C01780=1012.610,-71.664,-108.852,165.899,73.815,164.195
C01781=1012.611,-71.904,-108.833,165.879,73.747,164.164
C01782=1012.612,-72.145,-108.812,165.857,73.678,164.133
C01783=1012.613,-72.385,-108.791,165.837,73.609,164.102
C01784=1012.614,-72.626,-108.771,165.814,73.539,164.070
C01785=1012.614,-72.866,-108.751,165.795,73.470,164.040
C01786=1012.616,-73.107,-108.731,165.775,73.400,164.010
C01787=1012.617,-73.347,-108.710,165.755,73.330,163.979
C01788=1012.617,-73.587,-108.690,165.733,73.259,163.948
C01789=1012.618,-73.827,-108.669,165.715,73.188,163.919
C01790=1012.620,-74.067,-108.649,165.695,73.117,163.888
C01791=1012.621,-74.308,-108.628,165.674,73.045,163.858
C01792=1012.621,-74.547,-108.608,165.656,72.974,163.828
C01793=1012.623,-74.788,-108.588,165.638,72.901,163.799
C01794=1012.623,-75.027,-108.568,165.618,72.829,163.769
C01795=1012.624,-75.267,-108.547,165.599,72.756,163.739
C01796=1012.625,-75.507,-108.526,165.581,72.684,163.710
C01797=1012.627,-75.747,-108.507,165.563,72.611,163.680
C01798=1012.627,-75.987,-108.486,165.543,72.537,163.650
C01799=1012.629,-76.227,-108.465,165.527,72.463,163.622
C01800=1012.630,-76.466,-108.445,165.508,72.389,163.593
C01801=1012.631,-76.706,-108.424,165.491,72.314,163.564
C01802=1012.632,-76.945,-108.404,165.473,72.241,163.535
C01803=1012.633,-77.184,-108.384,165.456,72.165,163.506
C01804=1012.634,-77.424,-108.364,165.438,72.090,163.478
C01805=1012.635,-77.663,-108.344,165.423,72.014,163.450
C01806=1012.637,-77.902,-108.323,165.406,71.939,163.422
C01807=1012.637,-78.141,-108.303,165.390,71.863,163.394
C01808=1012.638,-78.380,-108.283,165.373,71.787,163.365
C01809=1012.640,-78.618,-108.262,165.357,71.711,163.338
C01810=1012.641,-78.857,-108.242,165.342,71.635,163.310
C01811=1012.642,-79.095,-108.222,165.326,71.557,163.282
C01812=1012.643,-79.334,-108.201,165.310,71.481,163.255
C01813=1012.644,-79.572,-108.182,165.296,71.403,163.228
C01814=1012.646,-79.810,-108.161,165.281,71.326,163.201
C01815=1012.647,-80.048,-108.141,165.266,71.248,163.173
C01816=1012.648,-80.341,-108.115,165.248,71.152,163.140
C01817=1012.651,-80.759,-108.080,165.223,71.014,163.093
C01818=1012.652,-80.996,-108.061,165.208,70.935,163.066
C01819=1012.653,-81.232,-108.040,165.194,70.856,163.039
C01820=1012.654,-81.468,-108.020,165.181,70.777,163.013
C01821=1012.656,-81.705,-108.000,165.168,70.698,162.987
C01822=1012.657,-81.943,-107.980,165.153,70.618,162.960
C01823=1012.658,-82.181,-107.959,165.140,70.538,162.934
C01824=1012.660,-82.418,-107.939,165.128,70.458,162.909
C01825=1012.661,-82.653,-107.919,165.116,70.378,162.883
C01826=1012.661,-82.889,-107.899,165.103,70.297,162.857
C01827=1012.664,-83.125,-107.879,165.090,70.217,162.832
C01828=1012.664,-83.361,-107.859,165.078,70.135,162.806
C01829=1012.665,-83.596,-107.840,165.066,70.055,162.781
C01830=1012.667,-83.829,-107.819,165.054,69.974,162.756
C01831=1012.668,-84.062,-107.799,165.043,69.893,162.731
C01832=1012.669,-84.295,-107.780,165.031,69.812,162.706
C01833=1012.671,-84.535,-107.759,165.019,69.728,162.680
C01834=1012.672,-84.792,-107.738,165.008,69.638,162.654
C01835=1012.674,-85.066,-107.714,164.994,69.542,162.625
C01836=1012.676,-85.351,-107.689,164.982,69.441,162.595
C01837=1012.678,-85.634,-107.666,164.969,69.341,162.565
C01838=1012.679,-85.904,-107.643,164.957,69.245,162.538
C01839=1012.681,-86.154,-107.622,164.947,69.156,162.512
C01840=1012.682,-86.389,-107.602,164.937,69.072,162.488
C01841=1012.683,-86.621,-107.582,164.927,68.988,162.464
C01842=1012.685,-86.849,-107.563,164.918,68.905,162.440
C01843=1012.686,-87.073,-107.544,164.910,68.825,162.418
C01844=1012.688,-87.293,-107.525,164.901,68.745,162.396
C01845=1012.689,-87.512,-107.506,164.893,68.665,162.373
C01846=1012.691,-87.727,-107.488,164.884,68.587,162.352
C01847=1012.692,-87.943,-107.470,164.875,68.508,162.329
C01848=1012.693,-88.170,-107.451,164.868,68.424,162.307
C01849=1012.695,-88.397,-107.431,164.860,68.341,162.285
C01850=1012.696,-88.630,-107.411,164.851,68.255,162.261
C01851=1012.698,-88.898,-107.389,164.842,68.156,162.235
C01852=1012.700,-89.194,-107.363,164.832,68.046,162.206
C01853=1012.702,-89.503,-107.337,164.822,67.931,162.175
C01854=1012.704,-89.803,-107.312,164.813,67.819,162.146
C01855=1012.706,-90.082,-107.288,164.804,67.714,162.119
C01856=1012.709,-90.479,-107.254,164.792,67.565,162.080
C01857=1012.711,-90.775,-107.230,164.784,67.452,162.052
C01858=1012.712,-91.025,-107.208,164.778,67.357,162.028
C01859=1012.714,-91.257,-107.188,164.771,67.268,162.006
C01860=1012.716,-91.488,-107.168,164.765,67.180,161.983
C01861=1012.717,-91.720,-107.149,164.760,67.091,161.962
C01862=1012.719,-91.951,-107.129,164.753,67.002,161.940
C01863=1012.721,-92.182,-107.110,164.748,66.913,161.918
C01864=1012.723,-92.412,-107.090,164.742,66.825,161.896
C01865=1012.724,-92.643,-107.070,164.738,66.735,161.875
C01866=1012.726,-92.873,-107.050,164.732,66.645,161.853
C01867=1012.728,-93.103,-107.032,164.726,66.556,161.831
C01868=1012.730,-93.333,-107.012,164.723,66.466,161.811
C01869=1012.731,-93.562,-106.992,164.718,66.377,161.790
C01870=1012.733,-93.790,-106.973,164.714,66.286,161.768
C01871=1012.734,-94.019,-106.953,164.709,66.197,161.747
C01872=1012.737,-94.326,-106.928,164.704,66.075,161.719
C01873=1012.740,-94.702,-106.896,164.697,65.926,161.685
C01874=1012.742,-94.928,-106.877,164.694,65.836,161.664
C01875=1012.743,-95.155,-106.858,164.691,65.746,161.644
C01876=1012.745,-95.381,-106.839,164.687,65.655,161.623
C01877=1012.746,-95.607,-106.819,164.684,65.565,161.604
C01878=1012.748,-95.832,-106.800,164.682,65.475,161.583
C01879=1012.750,-96.057,-106.780,164.679,65.384,161.563
C01880=1012.752,-96.281,-106.762,164.675,65.293,161.543
C01881=1012.754,-96.506,-106.743,164.673,65.203,161.523
C01882=1012.756,-96.730,-106.725,164.671,65.112,161.503
C01883=1012.758,-96.954,-106.705,164.669,65.021,161.484
C01884=1012.760,-97.178,-106.686,164.666,64.929,161.463
C01885=1012.761,-97.401,-106.667,164.664,64.838,161.444
C01886=1012.763,-97.625,-106.648,164.662,64.747,161.424
C01887=1012.766,-97.849,-106.629,164.662,64.655,161.405
C01888=1012.767,-98.072,-106.610,164.660,64.563,161.385
C01889=1012.769,-98.295,-106.591,164.658,64.471,161.366
C01890=1012.771,-98.520,-106.572,164.657,64.378,161.347
C01891=1012.773,-98.744,-106.554,164.655,64.285,161.327
C01892=1012.776,-98.967,-106.534,164.655,64.192,161.308
C01893=1012.777,-99.192,-106.516,164.654,64.099,161.289
C01894=1012.779,-99.416,-106.497,164.653,64.005,161.269
C01895=1012.781,-99.641,-106.477,164.654,63.911,161.251
C01896=1012.783,-99.867,-106.459,164.653,63.817,161.231
C01897=1012.784,-100.092,-106.440,164.653,63.722,161.212
C01898=1012.787,-100.318,-106.421,164.652,63.627,161.193
C01899=1012.789,-100.545,-106.402,164.652,63.532,161.173
C01900=1012.791,-100.771,-106.383,164.652,63.436,161.154
C01901=1012.793,-100.999,-106.364,164.653,63.340,161.135
C01902=1012.796,-101.226,-106.344,164.654,63.244,161.116
C01903=1012.798,-101.454,-106.325,164.655,63.147,161.097
C01904=1012.799,-101.682,-106.305,164.655,63.049,161.078
C01905=1012.802,-101.911,-106.287,164.656,62.952,161.059
C01906=1012.803,-102.140,-106.267,164.658,62.854,161.040
C01907=1012.806,-102.369,-106.248,164.658,62.756,161.021
C01908=1012.808,-102.598,-106.228,164.661,62.658,161.002
C01909=1012.810,-102.827,-106.209,164.661,62.559,160.983
C01910=1012.813,-103.057,-106.189,164.664,62.460,160.964
C01911=1012.814,-103.288,-106.171,164.666,62.361,160.946
C01912=1012.817,-103.517,-106.152,164.667,62.262,160.927
C01913=1012.819,-103.748,-106.132,164.669,62.161,160.908
C01914=1012.821,-103.979,-106.113,164.672,62.062,160.889
C01915=1012.823,-104.209,-106.093,164.674,61.961,160.870
C01916=1012.826,-104.440,-106.074,164.677,61.861,160.852
C01917=1012.829,-104.671,-106.054,164.679,61.760,160.833
C01918=1012.831,-104.902,-106.035,164.682,61.658,160.814
C01919=1012.833,-105.134,-106.016,164.685,61.557,160.796
C01920=1012.836,-105.365,-105.996,164.688,61.456,160.777
C01921=1012.838,-105.597,-105.976,164.693,61.354,160.759
C01922=1012.840,-105.828,-105.957,164.695,61.252,160.740
C01923=1012.842,-106.097,-105.935,164.699,61.134,160.719
C01924=1012.610,-133.983,-104.817,165.422,73.778,163.915
C01925=1012.608,-133.752,-104.837,165.458,73.892,163.966
C01926=1012.607,-133.521,-104.856,165.493,74.006,164.017
C01927=1012.606,-133.290,-104.874,165.530,74.120,164.069
C01928=1012.604,-133.059,-104.894,165.568,74.234,164.122
C01929=1012.602,-132.828,-104.912,165.606,74.346,164.176
C01930=1012.601,-132.597,-104.931,165.646,74.459,164.230
C01931=1012.600,-132.366,-104.949,165.685,74.573,164.284
C01932=1012.597,-132.135,-104.969,165.725,74.685,164.339
C01933=1012.597,-131.904,-104.988,165.766,74.797,164.395
C01934=1012.595,-131.674,-105.007,165.809,74.909,164.452
C01935=1012.594,-131.442,-105.025,165.851,75.020,164.509
C01936=1012.592,-131.211,-105.045,165.895,75.131,164.567
C01937=1012.591,-130.980,-105.063,165.940,75.243,164.626
C01938=1012.589,-130.750,-105.083,165.985,75.355,164.686
C01939=1012.588,-130.519,-105.101,166.032,75.465,164.747
C01940=1012.586,-130.288,-105.120,166.079,75.576,164.808
C01941=1012.585,-130.056,-105.139,166.127,75.687,164.870
C01942=1012.584,-129.825,-105.158,166.176,75.797,164.932
C01943=1012.583,-129.594,-105.177,166.225,75.906,164.996
C01944=1012.581,-129.247,-105.205,166.304,76.071,165.095
C01945=1012.579,-128.901,-105.234,166.382,76.235,165.193
C01946=1012.578,-128.670,-105.253,166.436,76.344,165.260
C01947=1012.576,-128.440,-105.272,166.492,76.453,165.329
C01948=1012.575,-128.208,-105.291,166.546,76.562,165.397
C01949=1012.574,-127.977,-105.310,166.603,76.670,165.467
C01950=1012.573,-127.746,-105.328,166.662,76.778,165.539
C01951=1012.571,-127.515,-105.348,166.722,76.886,165.612
C01952=1012.570,-127.284,-105.367,166.782,76.994,165.684
C01953=1012.569,-127.053,-105.386,166.845,77.102,165.760
C01954=1012.568,-126.822,-105.405,166.906,77.209,165.834
C01955=1012.567,-126.590,-105.424,166.970,77.317,165.911
C01956=1012.565,-126.360,-105.443,167.038,77.424,165.990
C01957=1012.564,-126.129,-105.462,167.104,77.531,166.069
C01958=1012.563,-125.898,-105.481,167.171,77.638,166.149
C01959=1012.562,-125.667,-105.501,167.239,77.743,166.229
C01960=1012.561,-125.435,-105.520,167.312,77.850,166.313
C01961=1012.559,-125.204,-105.538,167.384,77.955,166.397
C01962=1012.559,-124.973,-105.557,167.456,78.062,166.482
C01963=1012.558,-124.742,-105.576,167.532,78.168,166.570
C01964=1012.557,-124.511,-105.595,167.607,78.273,166.657
C01965=1012.556,-124.280,-105.614,167.687,78.379,166.748
C01966=1012.555,-124.050,-105.633,167.768,78.483,166.840
C01967=1012.554,-123.818,-105.652,167.849,78.588,166.933
C01968=1012.553,-123.587,-105.671,167.930,78.693,167.026
C01969=1012.552,-123.355,-105.690,168.017,78.798,167.124
C01970=1012.551,-123.125,-105.709,168.102,78.902,167.221
C01971=1012.550,-122.893,-105.728,168.191,79.006,167.321
C01972=1012.549,-122.662,-105.747,168.280,79.109,167.421
C01973=1012.548,-122.431,-105.767,168.372,79.214,167.524
C01974=1012.547,-122.200,-105.786,168.465,79.317,167.629
C01975=1012.546,-121.968,-105.804,168.561,79.420,167.735
C01976=1012.545,-121.737,-105.825,168.659,79.524,167.845
C01977=1012.543,-121.507,-105.843,168.760,79.627,167.956
C01978=1012.542,-121.275,-105.862,168.862,79.729,168.068
C01979=1012.542,-121.045,-105.882,168.968,79.832,168.185
C01980=1012.541,-120.813,-105.900,169.074,79.935,168.302
C01981=1012.540,-120.583,-105.920,169.185,80.037,168.422
C01982=1012.539,-120.351,-105.939,169.294,80.139,168.542
C01983=1012.539,-120.119,-105.958,169.410,80.241,168.668
C01984=1012.538,-119.888,-105.978,169.524,80.343,168.794
C01985=1012.537,-119.657,-105.996,169.644,80.444,168.923
C01986=1012.536,-119.426,-106.015,169.766,80.545,169.055
C01987=1012.535,-119.195,-106.035,169.889,80.646,169.188
C01988=1012.534,-118.963,-106.054,170.018,80.747,169.327
C01989=1012.533,-118.732,-106.073,170.147,80.847,169.466
C01990=1012.533,-118.501,-106.092,170.280,80.948,169.609
C01991=1012.531,-118.092,-106.126,170.523,81.125,169.870
C01992=1012.530,-117.807,-106.150,170.698,81.249,170.056
C01993=1012.529,-117.576,-106.169,170.847,81.348,170.215
C01994=1012.530,-117.345,-106.188,170.996,81.448,170.373
C01995=1012.529,-117.114,-106.206,171.150,81.547,170.537
C01996=1012.528,-116.883,-106.226,171.308,81.647,170.704
C01997=1012.527,-116.651,-106.245,171.467,81.745,170.872
C01998=1012.526,-116.420,-106.264,171.635,81.844,171.049
C01999=1012.526,-116.189,-106.284,171.803,81.942,171.227
C02000=1012.525,-115.958,-106.303,171.976,82.041,171.408
C02001=1012.524,-115.727,-106.322,172.154,82.139,171.596
C02002=1012.524,-115.495,-106.341,172.334,82.237,171.785
C02003=1012.523,-115.264,-106.361,172.524,82.334,171.983
C02004=1012.522,-115.033,-106.380,172.715,82.431,172.183
C02005=1012.522,-114.801,-106.399,172.911,82.529,172.388
C02006=1012.521,-114.570,-106.419,173.118,82.626,172.603
C02007=1012.520,-114.338,-106.437,173.323,82.722,172.817
C02008=1012.520,-114.107,-106.457,173.538,82.819,173.040
C02009=1012.519,-113.876,-106.476,173.759,82.916,173.270
C02010=1012.518,-113.645,-106.496,173.984,83.012,173.503
C02011=1012.518,-113.413,-106.515,174.216,83.107,173.743
C02012=1012.517,-113.181,-106.534,174.453,83.203,173.990
C02013=1012.517,-112.950,-106.554,174.700,83.298,174.245
C02014=1012.516,-112.719,-106.573,174.955,83.394,174.507
C02015=1012.515,-112.488,-106.592,175.212,83.488,174.773
C02016=1012.515,-112.256,-106.611,175.484,83.583,175.052
C02017=1012.515,-112.025,-106.630,175.758,83.677,175.335
C02018=1012.514,-111.793,-106.650,176.042,83.771,175.627
C02019=1012.514,-111.563,-106.669,176.336,83.865,175.928
C02020=1012.513,-111.330,-106.688,176.634,83.957,176.234
C02021=1012.512,-111.099,-106.707,176.948,84.051,176.556
C02022=1012.512,-110.868,-106.727,177.266,84.144,176.882
C02023=1012.511,-110.636,-106.746,177.597,84.236,177.220
C02024=1012.511,-110.405,-106.766,177.939,84.327,177.569
C02025=1012.511,-110.173,-106.785,178.292,84.420,177.931
C02026=1012.510,-109.942,-106.805,178.660,84.511,178.305
C02027=1012.510,-109.710,-106.824,179.033,84.602,178.686
C02028=1012.509,-109.479,-106.843,179.420,84.692,179.080
C02029=1012.509,-109.245,-106.863,179.828,84.783,179.496
C02030=1012.508,-109.004,-106.883,-179.733,84.876,179.941
C02031=1012.508,-108.754,-106.904,-179.271,84.972,-179.589
C02032=1012.508,-108.493,-106.926,-178.768,85.072,-179.077
C02033=1012.507,-108.225,-106.948,-178.225,85.174,-178.527
C02034=1012.507,-107.951,-106.971,-177.642,85.279,-177.936
C02035=1012.506,-107.674,-106.994,-177.040,85.382,-177.326
C02036=1012.505,-107.399,-107.017,-176.409,85.485,-176.686
C02037=1012.505,-107.129,-107.041,-175.756,85.585,-176.026
C02038=1012.505,-106.867,-107.062,-175.101,85.681,-175.363
C02039=1012.504,-106.614,-107.083,-174.437,85.773,-174.692
C02040=1012.504,-106.372,-107.104,-173.774,85.861,-174.022
C02041=1012.504,-106.136,-107.124,-173.103,85.946,-173.345
C02042=1012.503,-105.758,-107.155,-171.968,86.080,-172.200
C02043=1012.503,-105.442,-107.182,-170.971,86.189,-171.195
C02044=1012.503,-105.210,-107.201,-170.188,86.270,-170.405
C02045=1012.502,-104.979,-107.220,-169.382,86.349,-169.594
C02046=1012.502,-104.748,-107.240,-168.553,86.427,-168.758
C02047=1012.501,-104.516,-107.259,-167.673,86.504,-167.872
C02048=1012.501,-104.286,-107.278,-166.751,86.580,-166.944
C02049=1012.501,-104.054,-107.298,-165.803,86.655,-165.991
C02050=1012.502,-103.825,-107.318,-164.808,86.729,-164.990
C02051=1012.501,-103.594,-107.337,-163.769,86.801,-163.945
C02052=1012.500,-103.364,-107.356,-162.680,86.872,-162.851
C02053=1012.501,-103.134,-107.376,-161.552,86.943,-161.717
C02054=1012.499,-102.904,-107.395,-160.379,87.011,-160.538
C02055=1012.500,-102.675,-107.415,-159.145,87.078,-159.299
C02056=1012.500,-102.445,-107.434,-157.853,87.143,-158.001
C02057=1012.499,-102.216,-107.453,-156.504,87.207,-156.647
C02058=1012.499,-101.987,-107.473,-155.105,87.269,-155.242
C02059=1012.499,-101.759,-107.491,-153.627,87.329,-153.759
C02060=1012.499,-101.531,-107.511,-152.100,87.387,-152.227
C02061=1012.499,-101.303,-107.530,-150.532,87.442,-150.654
C02062=1012.499,-101.076,-107.550,-148.865,87.496,-148.982
C02063=1012.498,-100.849,-107.568,-147.155,87.547,-147.268
C02064=1012.499,-100.621,-107.587,-145.373,87.596,-145.481
C02065=1012.498,-100.396,-107.607,-143.518,87.642,-143.620
C02066=1012.498,-100.170,-107.626,-141.589,87.686,-141.687
C02067=1012.498,-99.944,-107.645,-139.610,87.726,-139.703
C02068=1012.498,-99.719,-107.664,-137.573,87.764,-137.661
C02069=1012.498,-99.494,-107.683,-135.467,87.798,-135.551
C02070=1012.498,-99.270,-107.701,-133.296,87.830,-133.376
C02071=1012.497,-99.045,-107.721,-131.089,87.858,-131.163
C02072=1012.497,-98.822,-107.740,-128.799,87.883,-128.869
C02073=1012.497,-98.597,-107.759,-126.499,87.904,-126.565
C02074=1012.497,-98.373,-107.778,-124.139,87.922,-124.200
C02075=1012.497,-98.150,-107.796,-121.757,87.935,-121.814
C02076=1012.497,-97.926,-107.815,-119.371,87.946,-119.424
C02077=1012.498,-97.703,-107.834,-116.939,87.953,-116.988
C02078=1012.497,-97.479,-107.853,-114.519,87.956,-114.563
C02079=1012.497,-97.256,-107.872,-112.071,87.955,-112.112
C02080=1012.497,-97.032,-107.891,-109.652,87.951,-109.688
C02081=1012.497,-96.808,-107.909,-107.246,87.943,-107.278
C02082=1012.497,-96.584,-107.929,-104.882,87.931,-104.911
C02083=1012.497,-96.360,-107.947,-102.528,87.916,-102.553
C02084=1012.496,-96.135,-107.967,-100.232,87.897,-100.252
C02085=1012.496,-95.910,-107.986,-97.978,87.875,-97.995
C02086=1012.497,-95.686,-108.005,-95.754,87.850,-95.767
C02087=1012.497,-95.460,-108.024,-93.602,87.822,-93.611
C02088=1012.497,-95.234,-108.044,-91.510,87.790,-91.516
C02089=1012.497,-95.007,-108.062,-89.460,87.756,-89.462
C02090=1012.497,-94.781,-108.081,-87.490,87.719,-87.488
C02091=1012.496,-94.553,-108.101,-85.584,87.679,-85.578
C02092=1012.497,-94.326,-108.120,-83.748,87.637,-83.739
C02093=1012.497,-94.098,-108.139,-81.974,87.592,-81.961
C02094=1012.497,-93.869,-108.158,-80.253,87.545,-80.237
C02095=1012.497,-93.641,-108.178,-78.611,87.496,-78.591
C02096=1012.496,-93.412,-108.198,-77.048,87.446,-77.026
C02097=1012.497,-93.182,-108.217,-75.532,87.393,-75.505
C02098=1012.497,-92.952,-108.237,-74.077,87.338,-74.047
C02099=1012.498,-92.598,-108.267,-71.951,87.251,-71.916
C02100=1012.497,-92.261,-108.295,-70.074,87.165,-70.034
C02101=1012.498,-92.030,-108.315,-68.844,87.104,-68.801
C02102=1012.497,-91.799,-108.334,-67.684,87.043,-67.639
C02103=1012.498,-91.568,-108.354,-66.554,86.980,-66.505
C02104=1012.497,-91.337,-108.374,-65.488,86.917,-65.436
C02105=1012.497,-91.105,-108.393,-64.449,86.851,-64.394
C02106=1012.498,-90.855,-108.414,-63.392,86.780,-63.334
C02107=1012.498,-90.558,-108.440,-62.190,86.694,-62.129
C02108=1012.498,-90.162,-108.474,-60.695,86.579,-60.628
C02109=1012.498,-89.884,-108.497,-59.706,86.496,-59.637
C02110=1012.498,-89.582,-108.523,-58.692,86.406,-58.619
C02111=1012.498,-89.274,-108.549,-57.706,86.313,-57.630
C02112=1012.499,-88.978,-108.574,-56.802,86.222,-56.722
C02113=1012.499,-88.710,-108.597,-56.028,86.140,-55.945
C02114=1012.500,-88.477,-108.617,-55.388,86.068,-55.302
C02115=1012.500,-88.251,-108.636,-54.781,85.998,-54.693
C02116=1012.499,-88.025,-108.655,-54.206,85.928,-54.116
C02117=1012.500,-87.808,-108.674,-53.669,85.860,-53.576
C02118=1012.500,-87.592,-108.692,-53.150,85.792,-53.055
C02119=1012.500,-87.373,-108.711,-52.646,85.723,-52.550
C02120=1012.501,-87.154,-108.730,-52.159,85.653,-52.061
C02121=1012.500,-86.931,-108.748,-51.673,85.582,-51.572
C02122=1012.500,-86.701,-108.768,-51.201,85.510,-51.098
C02123=1012.501,-86.470,-108.787,-50.737,85.436,-50.633
C02124=1012.501,-86.236,-108.808,-50.281,85.361,-50.174
C02125=1012.502,-85.985,-108.829,-49.812,85.281,-49.702
C02126=1012.502,-85.715,-108.852,-49.331,85.196,-49.219
C02127=1012.502,-85.433,-108.876,-48.840,85.105,-48.727
C02128=1012.502,-85.148,-108.900,-48.368,85.014,-48.252
C02129=1012.503,-84.872,-108.924,-47.926,84.925,-47.807
C02130=1012.503,-84.617,-108.945,-47.534,84.842,-47.414
C02131=1012.503,-84.376,-108.966,-47.173,84.765,-47.051
C02132=1012.503,-84.143,-108.986,-46.839,84.690,-46.715
C02133=1012.504,-83.911,-109.006,-46.514,84.616,-46.388
C02134=1012.504,-83.678,-109.026,-46.199,84.540,-46.072
C02135=1012.504,-83.443,-109.046,-45.892,84.465,-45.763
C02136=1012.504,-83.207,-109.066,-45.589,84.389,-45.459
C02137=1012.504,-82.970,-109.086,-45.299,84.313,-45.167
C02138=1012.505,-82.735,-109.106,-45.012,84.237,-44.878
C02139=1012.505,-82.499,-109.126,-44.737,84.161,-44.602
C02140=1012.505,-82.262,-109.146,-44.470,84.086,-44.333
C02141=1012.505,-82.025,-109.167,-44.209,84.010,-44.071
C02142=1012.506,-81.787,-109.186,-43.956,83.933,-43.816
C02143=1012.506,-81.551,-109.207,-43.709,83.857,-43.568
C02144=1012.507,-81.314,-109.226,-43.468,83.781,-43.326
C02145=1012.507,-81.078,-109.248,-43.237,83.705,-43.094
C02146=1012.508,-80.841,-109.267,-43.011,83.630,-42.867
C02147=1012.508,-80.604,-109.288,-42.787,83.554,-42.641
C02148=1012.508,-80.368,-109.308,-42.572,83.479,-42.426
C02149=1012.508,-80.130,-109.328,-42.363,83.403,-42.215
C02150=1012.508,-79.893,-109.348,-42.158,83.327,-42.010
C02151=1012.509,-79.654,-109.369,-41.958,83.253,-41.808
C02152=1012.509,-79.416,-109.389,-41.762,83.177,-41.612
C02153=1012.510,-79.178,-109.410,-41.575,83.102,-41.423
C02154=1012.510,-78.940,-109.430,-41.388,83.026,-41.236
C02155=1012.511,-78.701,-109.450,-41.209,82.951,-41.056
C02156=1012.511,-78.463,-109.470,-41.030,82.876,-40.876
C02157=1012.511,-78.223,-109.491,-40.858,82.801,-40.703
C02158=1012.511,-77.985,-109.511,-40.690,82.726,-40.535
C02159=1012.512,-77.746,-109.531,-40.525,82.651,-40.369
C02160=1012.512,-77.443,-109.557,-40.322,82.557,-40.165
C02161=1012.513,-77.029,-109.592,-40.054,82.428,-39.896
C02162=1012.513,-76.789,-109.613,-39.906,82.354,-39.747
C02163=1012.514,-76.550,-109.633,-39.760,82.280,-39.601
C02164=1012.514,-76.310,-109.654,-39.618,82.206,-39.458
C02165=1012.515,-76.071,-109.674,-39.478,82.132,-39.318
C02166=1012.515,-75.831,-109.695,-39.340,82.058,-39.179
C02167=1012.515,-75.590,-109.716,-39.205,81.984,-39.044
C02168=1012.516,-75.352,-109.736,-39.075,81.911,-38.914
C02169=1012.516,-75.111,-109.757,-38.945,81.838,-38.783
C02170=1012.516,-74.871,-109.777,-38.820,81.765,-38.658
C02171=1012.517,-74.631,-109.797,-38.698,81.692,-38.535
C02172=1012.517,-74.392,-109.818,-38.576,81.620,-38.413
C02173=1012.517,-74.151,-109.839,-38.458,81.546,-38.295
C02174=1012.518,-73.912,-109.859,-38.344,81.475,-38.181
C02175=1012.518,-73.671,-109.879,-38.229,81.402,-38.065
C02176=1012.519,-73.431,-109.900,-38.119,81.331,-37.955
C02177=1012.520,-73.191,-109.920,-38.011,81.259,-37.847
C02178=1012.519,-72.951,-109.941,-37.905,81.187,-37.741
C02179=1012.520,-72.710,-109.961,-37.801,81.115,-37.637
C02180=1012.520,-72.470,-109.982,-37.700,81.045,-37.536
C02181=1012.521,-72.230,-110.002,-37.598,80.973,-37.433
C02182=1012.522,-71.989,-110.023,-37.501,80.902,-37.337
C02183=1012.522,-71.748,-110.043,-37.405,80.831,-37.242
C02184=1012.522,-71.508,-110.064,-37.310,80.762,-37.145
C02185=1012.523,-71.267,-110.085,-37.217,80.691,-37.053
C02186=1012.523,-71.027,-110.106,-37.125,80.620,-36.962
C02187=1012.524,-70.787,-110.126,-37.037,80.551,-36.873
C02188=1012.525,-70.546,-110.146,-36.950,80.482,-36.786
C02189=1012.525,-70.305,-110.166,-36.861,80.412,-36.698
C02190=1012.525,-70.064,-110.187,-36.779,80.343,-36.617
C02191=1012.525,-69.824,-110.208,-36.696,80.274,-36.534
C02192=1012.526,-69.583,-110.229,-36.614,80.205,-36.452
C02193=1012.526,-69.343,-110.249,-36.535,80.137,-36.373
C02194=1012.527,-69.101,-110.270,-36.454,80.068,-36.292
C02195=1012.527,-68.861,-110.290,-36.378,79.999,-36.217
C02196=1012.528,-68.620,-110.310,-36.302,79.931,-36.142
C02197=1012.528,-68.380,-110.331,-36.229,79.865,-36.068
C02198=1012.529,-68.139,-110.352,-36.155,79.797,-35.995
C02199=1012.529,-67.899,-110.373,-36.085,79.729,-35.926
C02200=1012.529,-67.658,-110.393,-36.014,79.663,-35.855
C02201=1012.530,-67.417,-110.413,-35.944,79.596,-35.786
C02202=1012.531,-67.177,-110.433,-35.876,79.530,-35.718
C02203=1012.531,-66.936,-110.454,-35.808,79.463,-35.651
C02204=1012.531,-66.696,-110.475,-35.744,79.397,-35.587
C02205=1012.532,-66.455,-110.496,-35.677,79.331,-35.520
C02206=1012.533,-66.215,-110.516,-35.614,79.265,-35.458
C02207=1012.533,-65.976,-110.537,-35.553,79.201,-35.398
C02208=1012.533,-65.735,-110.557,-35.491,79.135,-35.336
C02209=1012.534,-65.495,-110.578,-35.429,79.070,-35.275
C02210=1012.534,-65.255,-110.598,-35.370,79.006,-35.217
C02211=1012.535,-65.016,-110.619,-35.311,78.942,-35.159
C02212=1012.535,-64.776,-110.639,-35.254,78.877,-35.103
C02213=1012.536,-64.536,-110.659,-35.199,78.814,-35.048
C02214=1012.536,-64.297,-110.680,-35.142,78.750,-34.992
C02215=1012.537,-64.058,-110.700,-35.088,78.687,-34.939
C02216=1012.537,-63.819,-110.720,-35.033,78.625,-34.884
C02217=1012.537,-63.580,-110.741,-34.980,78.562,-34.833
C02218=1012.538,-63.341,-110.762,-34.927,78.499,-34.780
C02219=1012.539,-63.102,-110.782,-34.877,78.437,-34.732
C02220=1012.539,-62.864,-110.802,-34.827,78.375,-34.682
C02221=1012.540,-62.625,-110.823,-34.777,78.313,-34.634
C02222=1012.540,-62.387,-110.843,-34.727,78.253,-34.584
C02223=1012.540,-62.149,-110.863,-34.679,78.191,-34.537
C02224=1012.541,-61.910,-110.884,-34.632,78.131,-34.490
C02225=1012.541,-61.673,-110.904,-34.585,78.070,-34.445
C02226=1012.542,-61.436,-110.924,-34.539,78.010,-34.399
C02227=1012.542,-61.198,-110.944,-34.494,77.950,-34.355
C02228=1012.543,-60.961,-110.964,-34.450,77.890,-34.313
C02229=1012.543,-60.724,-110.985,-34.405,77.831,-34.268
C02230=1012.544,-60.487,-111.005,-34.361,77.772,-34.225
C02231=1012.544,-60.250,-111.025,-34.318,77.713,-34.183
C02232=1012.545,-60.014,-111.045,-34.277,77.655,-34.143
C02233=1012.546,-59.778,-111.065,-34.235,77.597,-34.102
C02234=1012.546,-59.541,-111.085,-34.195,77.539,-34.064
C02235=1012.546,-59.305,-111.105,-34.155,77.481,-34.024
C02236=1012.547,-58.914,-111.139,-34.089,77.386,-33.960
C02237=1012.548,-58.599,-111.166,-34.037,77.310,-33.909
C02238=1012.548,-58.364,-111.186,-34.000,77.254,-33.873
C02239=1012.549,-58.129,-111.206,-33.963,77.197,-33.838
C02240=1012.549,-57.894,-111.226,-33.927,77.142,-33.803
C02241=1012.550,-57.659,-111.246,-33.890,77.086,-33.767
C02242=1012.550,-57.425,-111.266,-33.854,77.031,-33.732
C02243=1012.551,-57.190,-111.286,-33.819,76.976,-33.699
C02244=1012.551,-56.956,-111.306,-33.785,76.921,-33.665
C02245=1012.552,-56.722,-111.326,-33.750,76.866,-33.632
C02246=1012.552,-56.488,-111.346,-33.717,76.813,-33.600
C02247=1012.553,-56.254,-111.366,-33.682,76.758,-33.566
C02248=1012.553,-56.020,-111.385,-33.651,76.704,-33.536
C02249=1012.553,-55.786,-111.405,-33.618,76.650,-33.505
C02250=1012.554,-55.553,-111.425,-33.586,76.598,-33.474
C02251=1012.555,-55.319,-111.445,-33.554,76.545,-33.443
C02252=1012.554,-55.085,-111.465,-33.524,76.492,-33.415
C02253=1012.555,-54.851,-111.485,-33.493,76.440,-33.385
C02254=1012.556,-54.618,-111.505,-33.463,76.388,-33.355
///RCONF 0,0,0,0,1,0,0,0,0,0,0,0,0,0,0,0,0,0,0,0,0,0,0,0
C02255=1012.557,-54.384,-111.525,-33.432,76.336,-33.326
C02256=1012.556,-54.151,-111.545,-33.402,76.284,-33.297
C02257=1012.557,-53.917,-111.564,-33.374,76.233,-33.270
C02258=1012.558,-53.684,-111.584,-33.344,76.180,-33.242
C02259=1012.558,-53.450,-111.604,-33.315,76.130,-33.214
C02260=1012.559,-53.216,-111.625,-33.289,76.079,-33.189
C02261=1012.559,-52.982,-111.644,-33.260,76.029,-33.162
C02262=1012.560,-52.749,-111.664,-33.232,75.978,-33.135
C02263=1012.561,-52.515,-111.684,-33.206,75.928,-33.110
C02264=1012.560,-52.282,-111.704,-33.179,75.879,-33.085
C02265=1012.561,-52.048,-111.723,-33.153,75.829,-33.060
C02266=1012.561,-51.814,-111.743,-33.126,75.780,-33.034
C02267=1012.562,-51.581,-111.763,-33.100,75.731,-33.008
C02268=1012.562,-51.347,-111.784,-33.075,75.682,-32.986
C02269=1012.563,-51.113,-111.803,-33.051,75.634,-32.963
C02270=1012.564,-50.879,-111.823,-33.025,75.585,-32.937
C02271=1012.564,-50.646,-111.844,-33.000,75.536,-32.914
C02272=1012.564,-50.412,-111.863,-32.976,75.490,-32.891
C02273=1012.564,-50.179,-111.882,-32.952,75.441,-32.869
C02274=1012.565,-49.945,-111.902,-32.928,75.395,-32.846
C02275=1012.565,-49.711,-111.923,-32.906,75.347,-32.826
C02276=1012.566,-49.477,-111.942,-32.883,75.300,-32.804
C02277=1012.567,-49.244,-111.962,-32.859,75.253,-32.782
C02278=1012.567,-49.010,-111.983,-32.837,75.207,-32.760
C02279=1012.567,-48.776,-112.002,-32.814,75.162,-32.739
C02280=1012.568,-48.542,-112.022,-32.792,75.115,-32.717
C02281=1012.569,-48.309,-112.042,-32.770,75.070,-32.696
C02282=1012.569,-48.074,-112.062,-32.749,75.024,-32.677
C02283=1012.569,-47.842,-112.081,-32.728,74.979,-32.658
C02284=1012.570,-47.608,-112.101,-32.706,74.934,-32.638
C02285=1012.569,-47.374,-112.121,-32.686,74.890,-32.619
C02286=1012.570,-47.140,-112.141,-32.665,74.846,-32.599
C02287=1012.571,-46.907,-112.161,-32.645,74.801,-32.581
C02288=1012.571,-46.672,-112.181,-32.625,74.757,-32.562
C02289=1012.571,-46.439,-112.201,-32.605,74.713,-32.543
C02290=1012.572,-46.205,-112.221,-32.586,74.670,-32.525
C02291=1012.572,-45.971,-112.240,-32.565,74.627,-32.505
C02292=1012.573,-45.737,-112.260,-32.546,74.584,-32.488
C02293=1012.573,-45.503,-112.280,-32.527,74.541,-32.470
C02294=1012.573,-45.269,-112.300,-32.509,74.500,-32.453
C02295=1012.574,-45.036,-112.320,-32.490,74.457,-32.436
C02296=1012.575,-44.802,-112.339,-32.472,74.415,-32.419
C02297=1012.575,-44.568,-112.360,-32.454,74.374,-32.402
C02298=1012.575,-44.334,-112.379,-32.437,74.332,-32.387
C02299=1012.575,-44.100,-112.400,-32.418,74.291,-32.369
C02300=1012.576,-43.866,-112.419,-32.401,74.250,-32.352
C02301=1012.577,-43.632,-112.439,-32.384,74.209,-32.338
C02302=1012.576,-43.398,-112.459,-32.366,74.169,-32.320
C02303=1012.577,-43.164,-112.479,-32.349,74.128,-32.305
C02304=1012.578,-42.931,-112.499,-32.332,74.089,-32.289
C02305=1012.578,-42.696,-112.519,-32.317,74.050,-32.275
C02306=1012.579,-42.463,-112.538,-32.300,74.010,-32.259
C02307=1012.578,-42.228,-112.558,-32.284,73.971,-32.245
C02308=1012.579,-41.995,-112.578,-32.269,73.932,-32.231
C02309=1012.579,-41.760,-112.598,-32.252,73.894,-32.215
C02310=1012.579,-41.526,-112.617,-32.237,73.854,-32.202
C02311=1012.580,-41.293,-112.637,-32.221,73.816,-32.186
C02312=1012.581,-41.057,-112.657,-32.206,73.779,-32.173
C02313=1012.581,-40.824,-112.677,-32.191,73.741,-32.159
C02314=1012.581,-40.589,-112.697,-32.176,73.704,-32.146
C02315=1012.582,-40.356,-112.717,-32.162,73.666,-32.132
C02316=1012.582,-40.122,-112.737,-32.146,73.630,-32.117
C02317=1012.583,-39.888,-112.757,-32.132,73.592,-32.104
C02318=1012.583,-39.654,-112.776,-32.117,73.557,-32.091
C02319=1012.583,-39.419,-112.796,-32.104,73.520,-32.080
C02320=1012.584,-39.186,-112.816,-32.090,73.484,-32.067
C02321=1012.584,-38.951,-112.836,-32.076,73.448,-32.054
C02322=1012.585,-38.717,-112.856,-32.062,73.414,-32.041
C02323=1012.585,-38.483,-112.876,-32.049,73.378,-32.028
C02324=1012.585,-38.249,-112.895,-32.036,73.343,-32.017
C02325=1012.585,-38.015,-112.916,-32.022,73.308,-32.005
C02326=1012.586,-37.781,-112.935,-32.009,73.274,-31.992
C02327=1012.586,-37.547,-112.956,-31.996,73.240,-31.979
C02328=1012.586,-37.313,-112.975,-31.983,73.206,-31.969
C02329=1012.587,-37.078,-112.995,-31.970,73.172,-31.956
C02330=1012.587,-36.844,-113.015,-31.958,73.139,-31.946
C02331=1012.587,-36.610,-113.035,-31.946,73.105,-31.935
C02332=1012.588,-36.375,-113.054,-31.934,73.073,-31.924
C02333=1012.588,-36.142,-113.075,-31.921,73.040,-31.912
C02334=1012.588,-35.908,-113.094,-31.910,73.008,-31.903
C02335=1012.588,-35.673,-113.114,-31.898,72.975,-31.891
C02336=1012.589,-35.439,-113.134,-31.886,72.943,-31.880
C02337=1012.589,-35.204,-113.154,-31.874,72.912,-31.868
C02338=1012.590,-34.970,-113.173,-31.864,72.881,-31.860
C02339=1012.590,-34.736,-113.194,-31.851,72.850,-31.848
C02340=1012.590,-34.502,-113.213,-31.841,72.818,-31.839
C02341=1012.590,-34.268,-113.233,-31.830,72.788,-31.829
C02342=1012.591,-34.034,-113.253,-31.819,72.758,-31.818
C02343=1012.591,-33.799,-113.273,-31.808,72.727,-31.808
C02344=1012.591,-33.565,-113.293,-31.797,72.697,-31.798
C02345=1012.592,-33.331,-113.313,-31.787,72.667,-31.790
C02346=1012.591,-33.097,-113.332,-31.776,72.639,-31.779
C02347=1012.592,-32.863,-113.352,-31.766,72.609,-31.771
C02348=1012.592,-32.628,-113.371,-31.756,72.580,-31.761
C02349=1012.592,-32.395,-113.391,-31.745,72.551,-31.751
C02350=1012.592,-32.160,-113.411,-31.736,72.523,-31.744
C02351=1012.593,-31.925,-113.431,-31.725,72.495,-31.732
C02352=1012.593,-31.692,-113.451,-31.716,72.467,-31.724
C02353=1012.594,-31.457,-113.471,-31.706,72.439,-31.716
C02354=1012.594,-31.223,-113.490,-31.696,72.412,-31.706
C02355=1012.594,-30.989,-113.510,-31.688,72.384,-31.699
C02356=1012.594,-30.755,-113.530,-31.678,72.357,-31.689
C02357=1012.594,-30.521,-113.550,-31.668,72.331,-31.681
C02358=1012.595,-30.286,-113.569,-31.659,72.304,-31.672
C02359=1012.595,-30.053,-113.590,-31.650,72.278,-31.664
C02360=1012.595,-29.818,-113.609,-31.642,72.252,-31.658
C02361=1012.595,-29.583,-113.629,-31.633,72.226,-31.649
C02362=1012.596,-29.350,-113.649,-31.624,72.201,-31.641
C02363=1012.596,-29.134,-113.667,-31.616,72.178,-31.633
C02364=1012.597,-28.881,-113.688,-31.608,72.151,-31.626
C02365=1012.596,-28.647,-113.708,-31.599,72.126,-31.618
C02366=1012.596,-28.413,-113.729,-31.590,72.101,-31.610
C02367=1012.597,-28.179,-113.748,-31.583,72.077,-31.603
C02368=1012.597,-27.944,-113.768,-31.574,72.054,-31.595
C02369=1012.597,-27.711,-113.788,-31.567,72.030,-31.588
C02370=1012.597,-27.476,-113.808,-31.558,72.007,-31.580
C02371=1012.598,-27.242,-113.827,-31.551,71.983,-31.573
C02372=1012.597,-27.008,-113.847,-31.543,71.960,-31.567
C02373=1012.598,-26.774,-113.867,-31.535,71.937,-31.558
C02374=1012.598,-26.540,-113.886,-31.528,71.915,-31.552
C02375=1012.598,-26.305,-113.906,-31.520,71.892,-31.545
C02376=1012.599,-26.072,-113.926,-31.512,71.871,-31.537
C02377=1012.598,-25.837,-113.946,-31.506,71.849,-31.532
C02378=1012.599,-25.603,-113.965,-31.498,71.827,-31.524
C02379=1012.599,-25.369,-113.986,-31.492,71.806,-31.519
C02380=1012.599,-25.135,-114.005,-31.485,71.785,-31.512
C02381=1012.599,-24.901,-114.025,-31.478,71.764,-31.505
C02382=1012.599,-24.666,-114.045,-31.471,71.743,-31.498
C02383=1012.600,-24.433,-114.065,-31.464,71.724,-31.492
C02384=1012.599,-24.198,-114.085,-31.457,71.703,-31.485
C02385=1012.600,-23.964,-114.104,-31.451,71.683,-31.480
C02386=1012.600,-23.730,-114.124,-31.444,71.664,-31.473
C02387=1012.601,-23.496,-114.144,-31.438,71.646,-31.468
C02388=1012.600,-23.262,-114.163,-31.432,71.626,-31.463
C02389=1012.601,-23.028,-114.183,-31.425,71.607,-31.454
C02390=1012.600,-22.795,-114.203,-31.419,71.589,-31.449
C02391=1012.600,-22.560,-114.223,-31.413,71.570,-31.444
C02392=1012.601,-22.326,-114.242,-31.407,71.552,-31.439
C02393=1012.601,-22.092,-114.262,-31.401,71.534,-31.432
C02394=1012.601,-21.858,-114.282,-31.396,71.517,-31.428
C02395=1012.601,-21.624,-114.301,-31.389,71.499,-31.421
C02396=1012.602,-21.390,-114.321,-31.384,71.482,-31.416
C02397=1012.601,-21.156,-114.341,-31.378,71.466,-31.410
C02398=1012.601,-20.921,-114.361,-31.372,71.449,-31.405
C02399=1012.602,-20.688,-114.381,-31.368,71.433,-31.401
C02400=1012.601,-20.454,-114.401,-31.361,71.417,-31.394
C02401=1012.602,-20.176,-114.423,-31.355,71.398,-31.388
C02402=1012.602,-19.826,-114.453,-31.347,71.374,-31.380
C02403=1012.601,-19.565,-114.475,-31.342,71.358,-31.375
C02404=1012.602,-19.266,-114.501,-31.335,71.338,-31.368
C02405=1012.602,-18.940,-114.528,-31.329,71.317,-31.362
C02406=1012.602,-18.609,-114.557,-31.322,71.298,-31.356
C02407=1012.602,-18.291,-114.583,-31.316,71.279,-31.349
C02408=1012.602,-18.007,-114.607,-31.310,71.262,-31.344
C02409=1012.602,-17.759,-114.628,-31.305,71.249,-31.339
C02410=1012.602,-17.528,-114.648,-31.300,71.235,-31.333
C02411=1012.602,-17.297,-114.667,-31.297,71.223,-31.330
C02412=1012.602,-17.063,-114.686,-31.292,71.210,-31.326
C02413=1012.602,-16.826,-114.707,-31.288,71.197,-31.322
C02414=1012.602,-16.589,-114.726,-31.284,71.185,-31.317
C02415=1012.603,-16.354,-114.746,-31.279,71.173,-31.312
C02416=1012.603,-16.119,-114.766,-31.276,71.161,-31.309
C02417=1012.602,-15.883,-114.786,-31.271,71.150,-31.304
C02418=1012.602,-15.647,-114.806,-31.267,71.138,-31.300
C02419=1012.603,-15.414,-114.825,-31.263,71.127,-31.296
C02420=1012.602,-15.185,-114.845,-31.260,71.117,-31.293
C02421=1012.603,-14.957,-114.864,-31.256,71.106,-31.288
C02422=1012.603,-14.733,-114.883,-31.252,71.096,-31.284
C02423=1012.602,-14.510,-114.902,-31.249,71.087,-31.280
C02424=1012.602,-14.287,-114.921,-31.245,71.078,-31.276
C02425=1012.603,-14.063,-114.939,-31.242,71.069,-31.273
C02426=1012.603,-13.837,-114.959,-31.238,71.059,-31.268
C02427=1012.602,-13.608,-114.978,-31.235,71.051,-31.265
C02428=1012.603,-13.375,-114.998,-31.232,71.042,-31.262
C02429=1012.602,-13.138,-115.017,-31.229,71.033,-31.258
C02430=1012.602,-12.897,-115.038,-31.226,71.024,-31.255
C02431=1012.602,-12.652,-115.058,-31.223,71.015,-31.252
C02432=1012.602,-12.407,-115.079,-31.219,71.008,-31.247
C02433=1012.602,-12.160,-115.100,-31.216,70.999,-31.244
C02434=1012.603,-11.913,-115.120,-31.213,70.992,-31.241
C02435=1012.602,-11.666,-115.141,-31.210,70.983,-31.238
C02436=1012.601,-11.418,-115.162,-31.208,70.976,-31.234
C02437=1012.602,-11.169,-115.183,-31.205,70.968,-31.231
C02438=1012.602,-10.920,-115.204,-31.202,70.961,-31.227
C02439=1012.602,-10.671,-115.226,-31.198,70.955,-31.222
C02440=1012.601,-10.421,-115.247,-31.196,70.949,-31.220
C02441=1012.602,-10.171,-115.267,-31.193,70.943,-31.217
C02442=1012.601,-9.921,-115.289,-31.191,70.937,-31.215
C02443=1012.601,-9.669,-115.309,-31.189,70.931,-31.211
C02444=1012.601,-9.418,-115.331,-31.186,70.926,-31.207
C02445=1012.601,-9.167,-115.352,-31.183,70.920,-31.204
C02446=1012.601,-8.916,-115.373,-31.181,70.915,-31.201
C02447=1012.600,-8.665,-115.394,-31.179,70.911,-31.199
C02448=1012.601,-8.413,-115.416,-31.177,70.907,-31.195
C02449=1012.601,-8.161,-115.437,-31.175,70.902,-31.193
C02450=1012.600,-7.909,-115.458,-31.173,70.899,-31.191
C02451=1012.601,-7.655,-115.480,-31.171,70.895,-31.187
C02452=1012.600,-7.401,-115.500,-31.169,70.892,-31.184
C02453=1012.600,-7.146,-115.523,-31.167,70.889,-31.182
C02454=1012.600,-6.889,-115.544,-31.165,70.886,-31.179
C02455=1012.599,-6.633,-115.565,-31.163,70.883,-31.175
C02456=1012.600,-6.375,-115.587,-31.162,70.881,-31.174
C02457=1012.599,-6.117,-115.609,-31.160,70.879,-31.171
C02458=1012.599,-5.859,-115.630,-31.159,70.878,-31.168
C02459=1012.599,-5.601,-115.652,-31.158,70.876,-31.167
C02460=1012.599,-5.344,-115.674,-31.156,70.875,-31.163
C02461=1012.599,-5.092,-115.695,-31.155,70.874,-31.162
C02462=1012.598,-4.848,-115.716,-31.154,70.874,-31.160
C02463=1012.598,-4.613,-115.736,-31.153,70.873,-31.159
C02464=1012.598,-4.384,-115.754,-31.152,70.873,-31.156
C02465=1012.598,-4.158,-115.773,-31.150,70.873,-31.153
C02466=1012.598,-3.932,-115.793,-31.149,70.872,-31.151
C02467=1012.597,-3.702,-115.812,-31.149,70.873,-31.150
C02468=1012.597,-3.465,-115.833,-31.148,70.874,-31.148
C02469=1012.598,-3.222,-115.852,-31.147,70.875,-31.147
C02470=1012.597,-2.978,-115.873,-31.146,70.877,-31.143
C02471=1012.597,-2.733,-115.894,-31.146,70.878,-31.143
C02472=1012.597,-2.489,-115.914,-31.145,70.879,-31.141
C02473=1012.596,-2.246,-115.934,-31.145,70.882,-31.139
C02474=1012.597,-2.003,-115.955,-31.144,70.884,-31.138
C02475=1012.596,-1.761,-115.975,-31.144,70.887,-31.136
C02476=1012.595,-1.519,-115.996,-31.143,70.889,-31.134
C02477=1012.595,-1.279,-116.016,-31.143,70.892,-31.132
C02478=1012.595,-1.039,-116.037,-31.143,70.895,-31.131
C02479=1012.595,-0.800,-116.056,-31.143,70.899,-31.131
C02480=1012.594,-0.561,-116.076,-31.143,70.903,-31.129
C02481=1012.594,-0.323,-116.096,-31.143,70.906,-31.128
C02482=1012.594,-0.087,-116.116,-31.143,70.910,-31.126
C02483=1012.594,0.149,-116.136,-31.142,70.914,-31.124
C02484=1012.593,0.384,-116.156,-31.143,70.918,-31.125
C02485=1012.593,0.618,-116.175,-31.143,70.923,-31.123
C02486=1012.593,0.852,-116.195,-31.143,70.928,-31.122
C02487=1012.592,1.089,-116.215,-31.143,70.933,-31.119
C02488=1012.592,1.326,-116.235,-31.143,70.938,-31.119
C02489=1012.592,1.562,-116.255,-31.145,70.944,-31.119
C02490=1012.592,1.796,-116.274,-31.144,70.950,-31.117
C02491=1012.591,2.025,-116.294,-31.146,70.955,-31.118
C02492=1012.591,2.246,-116.313,-31.145,70.961,-31.115
C02493=1012.590,2.655,-116.346,-31.147,70.972,-31.115
C02494=1012.590,3.039,-116.379,-31.148,70.983,-31.113
C02495=1012.589,3.431,-116.412,-31.150,70.996,-31.113
C02496=1012.589,3.639,-116.430,-31.150,71.002,-31.112
C02497=1012.589,3.857,-116.448,-31.152,71.009,-31.112
C02498=1012.588,4.086,-116.467,-31.152,71.018,-31.111
C02499=1012.588,4.319,-116.486,-31.154,71.025,-31.111
C02500=1012.588,4.552,-116.507,-31.154,71.033,-31.110
C02501=1012.587,4.784,-116.526,-31.156,71.042,-31.110
C02502=1012.587,5.014,-116.545,-31.156,71.050,-31.109
C02503=1012.587,5.246,-116.564,-31.158,71.059,-31.109
C02504=1012.586,5.479,-116.584,-31.159,71.068,-31.109
C02505=1012.586,5.711,-116.603,-31.160,71.078,-31.108
C02506=1012.586,5.946,-116.623,-31.162,71.087,-31.108
C02507=1012.585,6.180,-116.643,-31.163,71.098,-31.108
C02508=1012.585,6.413,-116.663,-31.166,71.107,-31.109
C02509=1012.584,6.646,-116.682,-31.167,71.117,-31.108
C02510=1012.584,6.877,-116.701,-31.168,71.128,-31.107
C02511=1012.583,7.106,-116.721,-31.171,71.137,-31.109
C02512=1012.584,7.333,-116.740,-31.172,71.148,-31.109
C02513=1012.583,7.560,-116.758,-31.174,71.158,-31.109
C02514=1012.583,7.786,-116.777,-31.176,71.170,-31.110
C02515=1012.582,8.009,-116.796,-31.177,71.181,-31.108
C02516=1012.582,8.233,-116.815,-31.179,71.192,-31.108
C02517=1012.582,8.455,-116.834,-31.181,71.203,-31.110
C02518=1012.581,8.678,-116.853,-31.184,71.215,-31.111
C02519=1012.581,8.900,-116.871,-31.186,71.227,-31.111
C02520=1012.581,9.123,-116.890,-31.188,71.239,-31.110
C02521=1012.580,9.346,-116.909,-31.190,71.250,-31.112
C02522=1012.580,9.568,-116.927,-31.192,71.263,-31.111
C02523=1012.580,9.792,-116.946,-31.194,71.275,-31.112
C02524=1012.579,10.015,-116.965,-31.196,71.288,-31.112
C02525=1012.578,10.239,-116.984,-31.199,71.301,-31.113
C02526=1012.579,10.465,-117.003,-31.202,71.314,-31.114
C02527=1012.577,10.689,-117.022,-31.204,71.327,-31.115
C02528=1012.577,10.910,-117.041,-31.206,71.340,-31.115
C02529=1012.576,11.128,-117.058,-31.209,71.353,-31.116
C02530=1012.576,11.344,-117.076,-31.212,71.367,-31.119
C02531=1012.577,11.560,-117.095,-31.214,71.381,-31.118
C02532=1012.575,11.779,-117.113,-31.217,71.394,-31.119
C02533=1012.575,12.003,-117.132,-31.220,71.409,-31.120
C02534=1012.575,12.229,-117.151,-31.224,71.424,-31.122
C02535=1012.574,12.459,-117.170,-31.226,71.438,-31.123
C02536=1012.574,12.687,-117.189,-31.229,71.455,-31.124
C02537=1012.574,12.915,-117.209,-31.232,71.469,-31.125
C02538=1012.573,13.144,-117.228,-31.235,71.486,-31.126
C02539=1012.572,13.372,-117.248,-31.239,71.501,-31.128
C02540=1012.572,13.599,-117.266,-31.242,71.517,-31.129
C02541=1012.571,13.827,-117.285,-31.246,71.534,-31.131
C02542=1012.571,14.053,-117.304,-31.250,71.549,-31.133
C02543=1012.571,14.279,-117.323,-31.253,71.566,-31.134
C02544=1012.570,14.506,-117.342,-31.257,71.583,-31.136
C02545=1012.570,14.733,-117.361,-31.260,71.601,-31.137
C02546=1012.569,14.958,-117.380,-31.264,71.617,-31.139
C02547=1012.568,15.185,-117.399,-31.268,71.634,-31.141
C02548=1012.567,15.411,-117.418,-31.271,71.652,-31.142
C02549=1012.567,15.637,-117.437,-31.275,71.669,-31.144
C02550=1012.567,15.864,-117.456,-31.279,71.688,-31.146
C02551=1012.566,16.091,-117.474,-31.282,71.706,-31.147
C02552=1012.566,16.319,-117.494,-31.287,71.723,-31.150
C02553=1012.565,16.546,-117.514,-31.291,71.742,-31.153
C02554=1012.564,16.775,-117.533,-31.295,71.762,-31.154
C02555=1012.564,17.004,-117.552,-31.299,71.781,-31.156
C02556=1012.564,17.234,-117.571,-31.304,71.800,-31.159
C02557=1012.563,17.464,-117.590,-31.308,71.820,-31.160
C02558=1012.562,17.695,-117.610,-31.313,71.839,-31.164
C02559=1012.562,17.927,-117.629,-31.317,71.859,-31.166
C02560=1012.561,18.159,-117.648,-31.322,71.880,-31.169
C02561=1012.561,18.392,-117.668,-31.327,71.901,-31.171
C02562=1012.560,18.626,-117.688,-31.332,71.921,-31.175
C02563=1012.560,18.859,-117.707,-31.337,71.942,-31.178
C02564=1012.559,19.121,-117.730,-31.343,71.967,-31.181
C02565=1012.558,19.426,-117.755,-31.349,71.994,-31.184
C02566=1012.557,19.822,-117.787,-31.358,72.032,-31.190
C02567=1012.557,20.122,-117.813,-31.365,72.060,-31.194
C02568=1012.556,20.441,-117.840,-31.372,72.090,-31.198
C02569=1012.555,20.760,-117.866,-31.379,72.122,-31.202
C02570=1012.554,21.070,-117.893,-31.388,72.152,-31.207
C02571=1012.553,21.359,-117.917,-31.394,72.181,-31.212
C02572=1012.553,21.618,-117.939,-31.400,72.207,-31.215
C02573=1012.552,22.029,-117.973,-31.411,72.248,-31.222
C02574=1012.551,22.442,-118.008,-31.422,72.291,-31.228
C02575=1012.549,22.787,-118.036,-31.431,72.327,-31.235
C02576=1012.549,23.078,-118.061,-31.439,72.358,-31.241
C02577=1012.549,23.379,-118.086,-31.448,72.390,-31.246
C02578=1012.547,23.743,-118.116,-31.458,72.430,-31.253
C02579=1012.546,24.109,-118.147,-31.468,72.469,-31.259
C02580=1012.545,24.406,-118.172,-31.477,72.503,-31.265
C02581=1012.544,24.642,-118.192,-31.483,72.529,-31.268
C02582=1012.543,24.878,-118.212,-31.490,72.556,-31.273
C02583=1012.543,25.114,-118.231,-31.497,72.582,-31.278
C02584=1012.542,25.349,-118.251,-31.505,72.609,-31.283
C02585=1012.541,25.585,-118.271,-31.513,72.636,-31.290
C02586=1012.541,25.823,-118.291,-31.519,72.663,-31.293
C02587=1012.541,26.060,-118.311,-31.527,72.692,-31.298
C02588=1012.540,26.296,-118.331,-31.535,72.719,-31.305
C02589=1012.539,26.533,-118.350,-31.542,72.747,-31.310
C02590=1012.538,26.768,-118.369,-31.550,72.775,-31.315
C02591=1012.537,27.003,-118.390,-31.558,72.803,-31.320
C02592=1012.537,27.237,-118.409,-31.565,72.832,-31.325
C02593=1012.536,27.471,-118.429,-31.574,72.861,-31.332
C02594=1012.536,27.705,-118.448,-31.581,72.889,-31.337
C02595=1012.535,27.938,-118.468,-31.590,72.918,-31.344
C02596=1012.534,28.173,-118.488,-31.598,72.947,-31.349
C02597=1012.534,28.407,-118.507,-31.607,72.976,-31.356
C02598=1012.533,28.642,-118.526,-31.615,73.006,-31.361
C02599=1012.532,28.876,-118.547,-31.624,73.035,-31.368
C02600=1012.532,29.112,-118.566,-31.633,73.066,-31.375
C02601=1012.530,29.347,-118.586,-31.642,73.096,-31.381
C02602=1012.530,29.583,-118.605,-31.650,73.126,-31.387
C02603=1012.529,29.818,-118.625,-31.659,73.156,-31.394
C02604=1012.528,30.053,-118.645,-31.668,73.187,-31.401
C02605=1012.528,30.288,-118.664,-31.678,73.219,-31.408
C02606=1012.527,30.524,-118.684,-31.687,73.250,-31.415
C02607=1012.526,30.759,-118.703,-31.696,73.282,-31.422
C02608=1012.525,30.994,-118.724,-31.706,73.312,-31.429
C02609=1012.525,31.229,-118.743,-31.715,73.344,-31.436
C02610=1012.524,31.465,-118.763,-31.725,73.376,-31.443
C02611=1012.524,31.700,-118.782,-31.735,73.409,-31.451
C02612=1012.522,31.936,-118.802,-31.745,73.441,-31.459
C02613=1012.521,32.170,-118.822,-31.755,73.474,-31.467
C02614=1012.521,32.406,-118.842,-31.766,73.506,-31.476
C02615=1012.520,32.642,-118.862,-31.777,73.539,-31.485
C02616=1012.519,32.877,-118.881,-31.786,73.572,-31.491
C02617=1012.518,33.112,-118.900,-31.797,73.605,-31.500
C02618=1012.518,33.346,-118.920,-31.808,73.639,-31.509
C02619=1012.517,33.583,-118.940,-31.818,73.673,-31.516
C02620=1012.516,33.818,-118.960,-31.830,73.706,-31.526
C02621=1012.515,34.053,-118.979,-31.841,73.740,-31.535
C02622=1012.514,34.288,-118.999,-31.852,73.775,-31.545
C02623=1012.514,34.524,-119.018,-31.863,73.810,-31.552
C02624=1012.513,34.759,-119.039,-31.875,73.845,-31.562
C02625=1012.513,34.994,-119.058,-31.886,73.879,-31.571
C02626=1012.511,35.229,-119.078,-31.897,73.914,-31.579
C02627=1012.511,35.466,-119.098,-31.910,73.950,-31.591
C02628=1012.510,35.701,-119.117,-31.921,73.985,-31.599
C02629=1012.509,35.936,-119.136,-31.934,74.020,-31.610
C02630=1012.508,36.171,-119.156,-31.946,74.056,-31.620
C02631=1012.508,36.407,-119.176,-31.959,74.092,-31.630
C02632=1012.507,36.642,-119.196,-31.971,74.128,-31.640
C02633=1012.506,36.877,-119.215,-31.984,74.165,-31.652
C02634=1012.505,37.112,-119.235,-31.997,74.201,-31.662
C02635=1012.504,37.349,-119.255,-32.010,74.238,-31.672
C02636=1012.504,37.584,-119.274,-32.022,74.274,-31.682
C02637=1012.502,37.819,-119.294,-32.035,74.312,-31.693
C02638=1012.502,38.054,-119.313,-32.049,74.349,-31.705
C02639=1012.501,38.290,-119.333,-32.063,74.387,-31.717
C02640=1012.500,38.525,-119.353,-32.076,74.425,-31.728
C02641=1012.500,38.760,-119.373,-32.090,74.462,-31.738
C02642=1012.498,38.995,-119.392,-32.104,74.501,-31.751
C02643=1012.498,39.232,-119.412,-32.118,74.539,-31.763
C02644=1012.497,39.467,-119.431,-32.133,74.577,-31.776
C02645=1012.496,39.702,-119.451,-32.148,74.616,-31.789
C02646=1012.495,39.937,-119.470,-32.162,74.655,-31.800
C02647=1012.495,40.173,-119.490,-32.176,74.693,-31.813
C02648=1012.493,40.409,-119.510,-32.192,74.733,-31.826
C02649=1012.493,40.644,-119.529,-32.206,74.772,-31.838
C02650=1012.491,40.879,-119.549,-32.222,74.811,-31.853
C02651=1012.491,41.115,-119.569,-32.238,74.851,-31.866
C02652=1012.490,41.350,-119.588,-32.253,74.891,-31.879
C02653=1012.489,41.586,-119.608,-32.269,74.931,-31.893
C02654=1012.488,41.821,-119.628,-32.286,74.971,-31.908
C02655=1012.488,42.057,-119.647,-32.301,75.012,-31.920
C02656=1012.487,42.292,-119.667,-32.318,75.053,-31.936
C02657=1012.485,42.527,-119.687,-32.334,75.094,-31.950
C02658=1012.485,42.763,-119.707,-32.350,75.134,-31.964
C02659=1012.484,42.998,-119.726,-32.367,75.176,-31.979
C02660=1012.483,43.234,-119.746,-32.385,75.218,-31.995
C02661=1012.482,43.469,-119.765,-32.403,75.258,-32.011
C02662=1012.482,43.705,-119.785,-32.420,75.300,-32.026
C02663=1012.480,43.940,-119.805,-32.438,75.342,-32.042
C02664=1012.479,44.176,-119.825,-32.455,75.385,-32.057
C02665=1012.479,44.411,-119.844,-32.474,75.427,-32.074
C02666=1012.478,44.647,-119.864,-32.493,75.469,-32.091
C02667=1012.477,44.882,-119.884,-32.510,75.512,-32.107
C02668=1012.476,45.117,-119.903,-32.529,75.554,-32.124
C02669=1012.475,45.353,-119.923,-32.549,75.598,-32.141
C02670=1012.474,45.589,-119.942,-32.567,75.641,-32.157
C02671=1012.473,45.824,-119.961,-32.587,75.684,-32.177
C02672=1012.472,46.061,-119.981,-32.607,75.728,-32.195
C02673=1012.471,46.296,-120.001,-32.627,75.771,-32.213
C02674=1012.470,46.531,-120.020,-32.647,75.815,-32.231
C02675=1012.470,46.767,-120.040,-32.666,75.860,-32.248
C02676=1012.469,47.003,-120.060,-32.687,75.903,-32.267
C02677=1012.467,47.238,-120.079,-32.709,75.948,-32.287
C02678=1012.467,47.474,-120.099,-32.730,75.993,-32.306
C02679=1012.466,47.709,-120.118,-32.749,76.037,-32.324
C02680=1012.465,47.945,-120.138,-32.772,76.082,-32.345
C02681=1012.464,48.181,-120.158,-32.793,76.127,-32.364
C02682=1012.464,48.416,-120.177,-32.816,76.173,-32.386
C02683=1012.462,48.651,-120.197,-32.838,76.218,-32.406
C02684=1012.461,48.887,-120.217,-32.861,76.264,-32.428
C02685=1012.460,49.123,-120.236,-32.884,76.309,-32.448
C02686=1012.460,49.358,-120.255,-32.907,76.355,-32.471
C02687=1012.459,49.594,-120.275,-32.930,76.402,-32.491
C02688=1012.458,49.830,-120.295,-32.954,76.448,-32.514
C02689=1012.456,50.065,-120.315,-32.978,76.495,-32.536
C02690=1012.456,50.301,-120.334,-33.001,76.541,-32.557
C02691=1012.455,50.536,-120.354,-33.027,76.588,-32.583
C02692=1012.454,50.772,-120.374,-33.051,76.635,-32.604
C02693=1012.453,51.008,-120.394,-33.076,76.682,-32.628
C02694=1012.452,51.244,-120.412,-33.102,76.730,-32.653
C02695=1012.451,51.479,-120.432,-33.128,76.777,-32.677
C02696=1012.450,51.715,-120.452,-33.153,76.825,-32.700
C02697=1012.449,51.951,-120.472,-33.180,76.873,-32.725
C02698=1012.448,52.186,-120.491,-33.208,76.921,-32.753
C02699=1012.448,52.422,-120.511,-33.233,76.969,-32.776
C02700=1012.446,52.657,-120.531,-33.262,77.017,-32.804
C02701=1012.445,52.893,-120.550,-33.290,77.066,-32.830
C02702=1012.444,53.129,-120.570,-33.318,77.115,-32.857
C02703=1012.444,53.364,-120.589,-33.346,77.164,-32.884
C02704=1012.443,53.600,-120.609,-33.374,77.213,-32.911
C02705=1012.442,53.836,-120.629,-33.403,77.262,-32.938
C02706=1012.440,54.071,-120.648,-33.433,77.312,-32.968
C02707=1012.439,54.308,-120.668,-33.463,77.360,-32.996
C02708=1012.439,54.543,-120.687,-33.493,77.411,-33.024
C02709=1012.437,54.778,-120.706,-33.524,77.461,-33.055
C02710=1012.437,55.015,-120.727,-33.555,77.511,-33.084
C02711=1012.436,55.250,-120.746,-33.585,77.561,-33.113
C02712=1012.435,55.486,-120.765,-33.618,77.611,-33.144
C02713=1012.434,55.722,-120.785,-33.651,77.662,-33.176
C02714=1012.433,55.957,-120.804,-33.682,77.713,-33.207
C02715=1012.432,56.193,-120.825,-33.716,77.764,-33.240
C02716=1012.431,56.429,-120.844,-33.748,77.814,-33.271
C02717=1012.430,56.664,-120.863,-33.783,77.865,-33.304
C02718=1012.429,56.900,-120.883,-33.816,77.917,-33.336
C02719=1012.428,57.136,-120.902,-33.853,77.969,-33.372
C02720=1012.427,57.372,-120.923,-33.887,78.021,-33.405
C02721=1012.426,57.607,-120.942,-33.923,78.072,-33.440
C02722=1012.425,58.022,-120.976,-33.987,78.164,-33.502
C02723=1012.423,58.315,-121.000,-34.032,78.229,-33.546
C02724=1012.422,58.551,-121.021,-34.070,78.281,-33.583
C02725=1012.421,58.786,-121.040,-34.108,78.334,-33.620
C02726=1012.420,59.022,-121.059,-34.146,78.386,-33.658
C02727=1012.420,59.258,-121.079,-34.187,78.440,-33.698
C02728=1012.418,59.493,-121.098,-34.225,78.493,-33.735
C02729=1012.417,59.729,-121.118,-34.266,78.546,-33.776
C02730=1012.416,59.965,-121.137,-34.307,78.599,-33.816
C02731=1012.415,60.200,-121.157,-34.348,78.653,-33.856
C02732=1012.415,60.437,-121.177,-34.390,78.707,-33.897
C02733=1012.413,60.672,-121.196,-34.432,78.761,-33.938
C02734=1012.412,60.908,-121.215,-34.474,78.815,-33.980
C02735=1012.411,61.144,-121.235,-34.519,78.869,-34.025
C02736=1012.411,61.379,-121.255,-34.563,78.923,-34.067
C02737=1012.409,61.615,-121.274,-34.609,78.978,-34.113
C02738=1012.409,61.851,-121.294,-34.653,79.032,-34.157
C02739=1012.407,62.087,-121.313,-34.700,79.086,-34.204
C02740=1012.406,62.363,-121.337,-34.755,79.151,-34.257
C02741=1012.405,62.650,-121.360,-34.813,79.218,-34.315
C02742=1012.404,62.926,-121.383,-34.870,79.284,-34.373
C02743=1012.403,63.222,-121.408,-34.933,79.353,-34.435
C02744=1012.401,63.505,-121.431,-34.991,79.419,-34.492
C02745=1012.401,63.756,-121.452,-35.047,79.479,-34.548
C02746=1012.400,63.993,-121.472,-35.099,79.535,-34.600
C02747=1012.398,64.246,-121.493,-35.155,79.596,-34.655
C02748=1012.397,64.513,-121.514,-35.217,79.660,-34.717
C02749=1012.396,64.784,-121.537,-35.278,79.724,-34.778
C02750=1012.395,65.049,-121.559,-35.342,79.788,-34.842
C02751=1012.394,65.309,-121.581,-35.404,79.851,-34.904
C02752=1012.393,65.562,-121.601,-35.464,79.911,-34.963
C02753=1012.392,65.806,-121.622,-35.523,79.970,-35.022
C02754=1012.391,66.038,-121.641,-35.583,80.027,-35.083
C02755=1012.389,66.430,-121.674,-35.682,80.122,-35.181
C02756=1012.389,66.644,-121.691,-35.737,80.174,-35.237
C02757=1012.388,66.880,-121.711,-35.801,80.233,-35.300
C02758=1012.387,67.117,-121.730,-35.863,80.290,-35.363
C02759=1012.385,67.354,-121.750,-35.928,80.349,-35.427
C02760=1012.385,67.591,-121.770,-35.995,80.407,-35.495
C02761=1012.384,67.830,-121.790,-36.064,80.466,-35.564
C02762=1012.383,68.072,-121.810,-36.130,80.526,-35.630
C02763=1012.382,68.317,-121.830,-36.202,80.587,-35.702
C02764=1012.381,68.566,-121.851,-36.276,80.649,-35.777
C02765=1012.379,68.816,-121.871,-36.353,80.711,-35.855
C02766=1012.379,69.064,-121.892,-36.429,80.773,-35.931
C02767=1012.377,69.310,-121.912,-36.504,80.835,-36.006
C02768=1012.377,69.553,-121.933,-36.581,80.896,-36.084
C02769=1012.375,69.794,-121.952,-36.660,80.957,-36.163
C02770=1012.374,70.035,-121.972,-36.739,81.017,-36.244
C02771=1012.374,70.277,-121.992,-36.819,81.079,-36.323
C02772=1012.373,70.517,-122.012,-36.901,81.140,-36.406
C02773=1012.371,70.758,-122.032,-36.983,81.201,-36.488
C02774=1012.371,71.000,-122.053,-37.068,81.262,-36.574
C02775=1012.370,71.241,-122.072,-37.155,81.324,-36.661
C02776=1012.368,71.481,-122.092,-37.241,81.385,-36.748
C02777=1012.368,71.723,-122.112,-37.332,81.446,-36.840
C02778=1012.366,71.964,-122.132,-37.423,81.508,-36.932
C02779=1012.365,72.206,-122.152,-37.515,81.571,-37.024
C02780=1012.364,72.448,-122.172,-37.609,81.633,-37.119
C02781=1012.364,72.691,-122.192,-37.708,81.696,-37.220
C02782=1012.362,72.935,-122.212,-37.807,81.759,-37.320
C02783=1012.361,73.180,-122.233,-37.908,81.822,-37.421
C02784=1012.361,73.424,-122.253,-38.010,81.886,-37.525
C02785=1012.360,73.670,-122.273,-38.117,81.950,-37.633
C02786=1012.358,73.917,-122.293,-38.225,82.014,-37.742
C02787=1012.358,74.168,-122.314,-38.335,82.079,-37.852
C02788=1012.356,74.435,-122.336,-38.459,82.150,-37.978
C02789=1012.355,74.707,-122.359,-38.585,82.220,-38.106
C02790=1012.354,74.965,-122.380,-38.709,82.289,-38.230
C02791=1012.353,75.214,-122.401,-38.830,82.354,-38.354
C02792=1012.352,75.462,-122.421,-38.954,82.419,-38.479
C02793=1012.351,75.708,-122.442,-39.077,82.483,-38.603
C02794=1012.350,75.952,-122.462,-39.205,82.548,-38.733
C02795=1012.349,76.193,-122.482,-39.329,82.612,-38.857
C02796=1012.348,76.431,-122.502,-39.459,82.675,-38.990
C02797=1012.347,76.666,-122.521,-39.589,82.738,-39.121
C02798=1012.346,76.900,-122.540,-39.717,82.800,-39.250
C02799=1012.345,77.130,-122.560,-39.849,82.860,-39.384
C02800=1012.344,77.359,-122.579,-39.983,82.921,-39.520
C02801=1012.344,77.586,-122.597,-40.120,82.982,-39.658
C02802=1012.343,77.814,-122.616,-40.258,83.044,-39.797
C02803=1012.342,78.041,-122.635,-40.400,83.104,-39.941
C02804=1012.341,78.270,-122.654,-40.544,83.165,-40.087
C02805=1012.340,78.500,-122.673,-40.694,83.227,-40.239
C02806=1012.339,78.733,-122.692,-40.847,83.289,-40.393
C02807=1012.338,78.967,-122.712,-41.006,83.353,-40.554
C02808=1012.337,79.205,-122.732,-41.168,83.416,-40.718
C02809=1012.336,79.444,-122.751,-41.336,83.481,-40.888
C02810=1012.335,79.686,-122.771,-41.512,83.546,-41.066
C02811=1012.334,79.931,-122.791,-41.691,83.613,-41.247
C02812=1012.333,80.304,-122.822,-41.978,83.713,-41.537
C02813=1012.332,80.649,-122.850,-42.251,83.806,-41.814
C02814=1012.331,80.866,-122.868,-42.423,83.865,-41.987
C02815=1012.330,81.084,-122.886,-42.602,83.924,-42.168
C02816=1012.329,81.313,-122.905,-42.799,83.986,-42.367
C02817=1012.328,81.555,-122.925,-43.011,84.052,-42.582
C02818=1012.327,81.802,-122.946,-43.227,84.119,-42.800
C02819=1012.326,82.050,-122.966,-43.454,84.186,-43.029
C02820=1012.325,82.296,-122.987,-43.686,84.253,-43.265
C02821=1012.324,82.542,-123.008,-43.924,84.320,-43.505
C02822=1012.323,82.788,-123.028,-44.168,84.387,-43.752
C02823=1012.322,83.033,-123.048,-44.412,84.454,-43.998
///RCONF 0,0,0,0,0,0,0,0,0,0,0,0,0,0,0,0,0,0,0,0,0,0,0,0
C02824=1012.321,83.279,-123.068,-44.668,84.520,-44.256
C02825=1012.320,83.525,-123.088,-44.930,84.587,-44.521
C02826=1012.319,83.769,-123.109,-45.199,84.654,-44.793
C02827=1012.318,84.012,-123.128,-45.475,84.720,-45.072
C02828=1012.317,84.257,-123.149,-45.758,84.786,-45.358
C02829=1012.317,84.500,-123.169,-46.049,84.852,-45.652
C02830=1012.315,84.742,-123.189,-46.347,84.918,-45.953
C02831=1012.314,84.984,-123.209,-46.654,84.984,-46.263
C02832=1012.313,85.226,-123.229,-46.968,85.050,-46.580
C02833=1012.313,85.467,-123.249,-47.292,85.116,-46.906
C02834=1012.312,85.708,-123.269,-47.624,85.181,-47.242
C02835=1012.311,85.948,-123.289,-47.966,85.246,-47.587
C02836=1012.311,86.188,-123.309,-48.317,85.311,-47.942
C02837=1012.310,86.428,-123.328,-48.679,85.375,-48.306
C02838=1012.309,86.667,-123.348,-49.051,85.440,-48.682
C02839=1012.308,86.906,-123.368,-49.434,85.505,-49.067
C02840=1012.307,87.143,-123.388,-49.820,85.568,-49.457
C02841=1012.306,87.380,-123.408,-50.226,85.632,-49.866
C02842=1012.305,87.613,-123.426,-50.636,85.694,-50.280
C02843=1012.304,87.844,-123.446,-51.058,85.756,-50.705
C02844=1012.303,88.071,-123.465,-51.476,85.816,-51.126
C02845=1012.302,88.296,-123.483,-51.915,85.876,-51.569
C02846=1012.301,88.520,-123.502,-52.358,85.935,-52.015
C02847=1012.300,88.743,-123.520,-52.814,85.994,-52.475
C02848=1012.300,88.969,-123.539,-53.286,86.053,-52.949
C02849=1012.299,89.196,-123.558,-53.789,86.113,-53.457
C02850=1012.299,89.425,-123.576,-54.299,86.172,-53.970
C02851=1012.298,89.658,-123.596,-54.846,86.233,-54.521
C02852=1012.297,89.894,-123.615,-55.414,86.295,-55.092
C02853=1012.296,90.178,-123.638,-56.131,86.367,-55.815
C02854=1012.295,90.512,-123.667,-57.002,86.453,-56.690
C02855=1012.293,90.831,-123.693,-57.886,86.534,-57.580
C02856=1012.292,91.090,-123.714,-58.633,86.599,-58.332
C02857=1012.291,91.326,-123.734,-59.331,86.657,-59.033
C02858=1012.291,91.562,-123.754,-60.068,86.716,-59.774
C02859=1012.290,91.797,-123.773,-60.828,86.774,-60.538
C02860=1012.289,92.032,-123.792,-61.616,86.831,-61.331
C02861=1012.288,92.267,-123.812,-62.437,86.888,-62.156
C02862=1012.287,92.503,-123.831,-63.284,86.943,-63.007
C02863=1012.287,92.738,-123.850,-64.167,86.999,-63.895
C02864=1012.286,92.974,-123.871,-65.079,87.053,-64.811
C02865=1012.285,93.209,-123.890,-66.030,87.107,-65.766
C02866=1012.284,93.444,-123.909,-67.031,87.161,-66.772
C02867=1012.284,93.679,-123.928,-68.057,87.213,-67.802
C02868=1012.282,93.915,-123.948,-69.121,87.265,-68.870
C02869=1012.282,94.150,-123.967,-70.241,87.315,-69.995
C02870=1012.282,94.386,-123.987,-71.388,87.364,-71.146
C02871=1012.281,94.620,-124.007,-72.594,87.413,-72.357
C02872=1012.280,94.855,-124.026,-73.845,87.460,-73.614
C02873=1012.279,95.091,-124.046,-75.153,87.506,-74.926
C02874=1012.278,95.326,-124.065,-76.483,87.551,-76.260
C02875=1012.277,95.561,-124.085,-77.878,87.594,-77.661
C02876=1012.277,95.797,-124.104,-79.334,87.636,-79.122
C02877=1012.276,96.033,-124.124,-80.843,87.677,-80.635
C02878=1012.275,96.268,-124.143,-82.391,87.715,-82.189
C02879=1012.274,96.503,-124.163,-84.024,87.752,-83.826
C02880=1012.273,96.738,-124.182,-85.690,87.787,-85.498
C02881=1012.273,96.973,-124.201,-87.408,87.821,-87.221
C02882=1012.272,97.209,-124.221,-89.198,87.852,-89.017
C02883=1012.272,97.444,-124.241,-91.019,87.881,-90.842
C02884=1012.271,97.679,-124.261,-92.887,87.908,-92.715
C02885=1012.270,97.914,-124.280,-94.822,87.932,-94.656
C02886=1012.269,98.150,-124.300,-96.821,87.955,-96.660
C02887=1012.268,98.385,-124.319,-98.819,87.974,-98.664
C02888=1012.268,98.620,-124.338,-100.896,87.991,-100.746
C02889=1012.266,99.005,-124.370,-104.318,88.013,-104.177
C02890=1012.266,99.326,-124.397,-107.255,88.026,-107.122
C02891=1012.265,99.561,-124.417,-109.429,88.032,-109.301
C02892=1012.264,99.796,-124.436,-111.612,88.036,-111.490
C02893=1012.263,100.031,-124.455,-113.799,88.036,-113.683
C02894=1012.263,100.267,-124.475,-115.983,88.034,-115.873
C02895=1012.262,100.502,-124.495,-118.158,88.028,-118.053
C02896=1012.261,100.738,-124.514,-120.335,88.020,-120.237
C02897=1012.261,100.972,-124.534,-122.471,88.009,-122.379
C02898=1012.260,101.207,-124.553,-124.606,87.995,-124.519
C02899=1012.259,101.442,-124.572,-126.699,87.978,-126.618
C02900=1012.259,101.679,-124.592,-128.737,87.959,-128.663
C02901=1012.258,101.914,-124.612,-130.775,87.937,-130.706
C02902=1012.258,102.149,-124.631,-132.740,87.912,-132.678
C02903=1012.257,102.383,-124.651,-134.667,87.885,-134.611
C02904=1012.256,102.619,-124.670,-136.557,87.856,-136.506
C02905=1012.255,102.854,-124.689,-138.391,87.824,-138.347
C02906=1012.255,103.090,-124.709,-140.170,87.790,-140.132
C02907=1012.254,103.325,-124.729,-141.892,87.754,-141.861
C02908=1012.253,103.560,-124.749,-143.557,87.716,-143.532
C02909=1012.253,103.795,-124.768,-145.164,87.676,-145.146
C02910=1012.252,104.030,-124.787,-146.715,87.634,-146.704
C02911=1012.251,104.266,-124.807,-148.210,87.590,-148.205
C02912=1012.251,104.500,-124.827,-149.650,87.545,-149.652
C02913=1012.251,104.735,-124.846,-151.057,87.498,-151.065
C02914=1012.249,104.971,-124.866,-152.397,87.450,-152.412
C02915=1012.249,105.206,-124.885,-153.698,87.400,-153.719
C02916=1012.248,105.441,-124.904,-154.929,87.349,-154.958
C02917=1012.248,105.676,-124.925,-156.137,87.297,-156.173
C02918=1012.247,105.912,-124.944,-157.292,87.243,-157.334
C02919=1012.247,106.147,-124.963,-158.406,87.188,-158.455
C02920=1012.246,106.382,-124.983,-159.476,87.132,-159.532
C02921=1012.245,106.616,-125.003,-160.499,87.076,-160.562
C02922=1012.245,106.852,-125.022,-161.486,87.018,-161.557
C02923=1012.244,107.088,-125.042,-162.435,86.959,-162.513
C02924=1012.244,107.322,-125.062,-163.345,86.899,-163.431
C02925=1012.243,107.557,-125.081,-164.218,86.840,-164.310
C02926=1012.243,107.793,-125.101,-165.074,86.778,-165.173
C02927=1012.242,108.028,-125.120,-165.883,86.716,-165.990
C02928=1012.242,108.263,-125.140,-166.674,86.653,-166.788
C02929=1012.241,108.498,-125.160,-167.422,86.590,-167.544
C02930=1012.240,108.733,-125.179,-168.157,86.526,-168.286
C02931=1012.240,108.968,-125.199,-168.862,86.461,-168.999
C02932=1012.240,109.204,-125.218,-169.540,86.396,-169.685
C02933=1012.239,109.439,-125.238,-170.194,86.330,-170.346
C02934=1012.238,109.674,-125.257,-170.824,86.264,-170.983
C02935=1012.238,109.909,-125.277,-171.432,86.197,-171.599
C02936=1012.237,110.145,-125.297,-172.016,86.130,-172.192
C02937=1012.236,110.380,-125.316,-172.581,86.062,-172.765
C02938=1012.236,110.614,-125.336,-173.126,85.994,-173.317
C02939=1012.236,110.850,-125.355,-173.662,85.925,-173.861
C02940=1012.235,111.085,-125.375,-174.169,85.857,-174.376
C02941=1012.235,111.320,-125.395,-174.668,85.787,-174.884
C02942=1012.234,111.555,-125.414,-175.141,85.717,-175.365
C02943=1012.234,111.791,-125.434,-175.608,85.647,-175.839
C02944=1012.233,112.025,-125.454,-176.049,85.577,-176.289
C02945=1012.233,112.260,-125.473,-176.485,85.506,-176.734
C02946=1012.232,112.496,-125.492,-176.907,85.435,-177.164
C02947=1012.232,112.731,-125.513,-177.315,85.363,-177.580
C02948=1012.231,112.966,-125.532,-177.710,85.292,-177.984
C02949=1012.231,113.201,-125.552,-178.092,85.220,-178.374
C02950=1012.230,113.437,-125.572,-178.471,85.147,-178.761
C02951=1012.230,113.672,-125.591,-178.829,85.075,-179.128
C02952=1012.230,113.906,-125.611,-179.176,85.002,-179.484
C02953=1012.230,114.142,-125.630,-179.521,84.929,-179.837
C02954=1012.228,114.377,-125.650,-179.847,84.856,179.828
C02955=1012.228,114.612,-125.670,179.830,84.782,179.496
C02956=1012.228,114.847,-125.689,179.523,84.709,179.180
C02957=1012.228,115.082,-125.709,179.218,84.635,178.866
C02958=1012.227,115.317,-125.729,178.922,84.560,178.562
C02959=1012.226,115.553,-125.748,178.635,84.486,178.266
C02960=1012.226,115.788,-125.768,178.356,84.411,177.978
C02961=1012.226,116.023,-125.787,178.085,84.337,177.698
C02962=1012.225,116.335,-125.814,177.736,84.237,177.337
C02963=1012.225,116.728,-125.847,177.312,84.111,176.897
C02964=1012.224,116.963,-125.866,177.071,84.035,176.647
C02965=1012.223,117.199,-125.886,176.830,83.960,176.397
C02966=1012.223,117.433,-125.906,176.602,83.884,176.159
C02967=1012.223,117.669,-125.926,176.374,83.808,175.922
C02968=1012.223,117.904,-125.945,176.158,83.732,175.696
C02969=1012.222,118.139,-125.965,175.943,83.656,175.471
C02970=1012.222,118.374,-125.985,175.733,83.579,175.252
C02971=1012.222,118.609,-126.004,175.528,83.502,175.038
C02972=1012.221,118.844,-126.024,175.329,83.426,174.829
C02973=1012.221,119.080,-126.044,175.136,83.349,174.625
C02974=1012.220,119.315,-126.063,174.947,83.272,174.426
C02975=1012.220,119.550,-126.084,174.757,83.194,174.228
C02976=1012.220,119.785,-126.103,174.578,83.117,174.039
C02977=1012.220,120.020,-126.123,174.403,83.040,173.854
C02978=1012.219,120.256,-126.143,174.229,82.962,173.669
C02979=1012.219,120.490,-126.162,174.058,82.884,173.489
C02980=1012.219,120.726,-126.182,173.896,82.807,173.317
C02981=1012.219,120.960,-126.202,173.741,82.732,173.151
C02982=1012.218,121.196,-126.223,173.595,82.660,172.996
C02983=1012.218,121.431,-126.242,173.452,82.589,172.844
C02984=1012.217,121.666,-126.262,173.313,82.516,172.695
C02985=1012.217,121.901,-126.282,173.176,82.445,172.549
C02986=1012.217,122.136,-126.303,173.043,82.372,172.407
C02987=1012.216,122.371,-126.322,172.914,82.300,172.267
C02988=1012.216,122.607,-126.342,172.787,82.228,172.130
C02989=1012.215,122.841,-126.363,172.658,82.155,171.992
C02990=1012.216,123.077,-126.383,172.536,82.083,171.860
C02991=1012.216,123.312,-126.403,172.413,82.010,171.727
C02992=1012.215,123.547,-126.423,172.296,81.938,171.601
C02993=1012.215,123.782,-126.443,172.179,81.865,171.473
C02994=1012.214,124.017,-126.464,172.065,81.791,171.349
C02995=1012.214,124.253,-126.483,171.952,81.718,171.226
C02996=1012.213,124.488,-126.503,171.842,81.645,171.106
C02997=1012.214,124.723,-126.524,171.733,81.571,170.988
C02998=1012.214,124.958,-126.544,171.628,81.498,170.872
C02999=1012.213,125.193,-126.564,171.525,81.424,170.759
C03000=1012.213,125.428,-126.584,171.424,81.351,170.647
C03001=1012.212,125.663,-126.604,171.321,81.277,170.534
C03002=1012.213,125.898,-126.624,171.225,81.204,170.428
C03003=1012.213,126.134,-126.645,171.126,81.130,170.319
C03004=1012.212,126.369,-126.664,171.034,81.056,170.216
C03005=1012.212,126.604,-126.685,170.939,80.982,170.111
C03006=1012.212,126.840,-126.705,170.848,80.907,170.008
C03007=1012.211,127.074,-126.725,170.757,80.834,169.907
C03008=1012.212,127.309,-126.745,170.669,80.759,169.809
C03009=1012.211,127.545,-126.765,170.581,80.685,169.711
C03010=1012.211,127.780,-126.785,170.497,80.611,169.615
C03011=1012.211,128.015,-126.805,170.414,80.536,169.522
C03012=1012.211,128.250,-126.826,170.333,80.462,169.430
C03013=1012.211,128.485,-126.846,170.253,80.388,169.339
C03014=1012.210,128.721,-126.866,170.172,80.313,169.247
C03015=1012.210,128.956,-126.886,170.096,80.238,169.159
C03016=1012.210,129.191,-126.906,170.018,80.163,169.071
C03017=1012.210,129.426,-126.927,169.945,80.088,168.986
C03018=1012.210,129.661,-126.947,169.870,80.013,168.901
C03019=1012.209,129.896,-126.968,169.797,79.938,168.816
C03020=1012.209,130.132,-126.987,169.725,79.863,168.733
C03021=1012.209,130.367,-127.007,169.655,79.788,168.652
C03022=1012.209,130.602,-127.028,169.586,79.712,168.572
C03023=1012.209,130.837,-127.048,169.519,79.637,168.493
C03024=1012.208,131.072,-127.069,169.452,79.562,168.415
C03025=1012.209,131.308,-127.089,169.387,79.487,168.339
C03026=1012.209,131.543,-127.108,169.321,79.411,168.261
C03027=1012.208,131.778,-127.129,169.260,79.335,168.188
C03028=1012.208,132.013,-127.149,169.196,79.260,168.113
C03029=1012.209,132.248,-127.169,169.136,79.185,168.041
C03030=1012.208,132.484,-127.190,169.075,79.109,167.968
C03031=1012.209,132.719,-127.210,169.016,79.032,167.897
C03032=1012.208,132.954,-127.231,168.957,78.957,167.827
C03033=1012.208,133.190,-127.250,168.900,78.880,167.758
C03034=1012.208,133.425,-127.270,168.843,78.805,167.689
C03035=1012.208,133.782,-127.301,168.759,78.689,167.588
C03036=1012.208,134.131,-127.332,168.682,78.576,167.491
C03037=1012.207,134.365,-127.352,168.627,78.500,167.425
C03038=1012.208,134.601,-127.372,168.577,78.424,167.362
C03039=1012.207,134.840,-127.392,168.524,78.345,167.297
C03040=1012.207,135.136,-127.419,168.459,78.249,167.218
C03041=1012.208,135.422,-127.442,168.401,78.157,167.144
C03042=1012.208,135.655,-127.463,168.352,78.081,167.083
C03043=1012.207,135.879,-127.482,168.309,78.008,167.028
C03044=1012.208,136.298,-127.518,168.227,77.871,166.923
C03045=1012.208,136.684,-127.552,168.153,77.745,166.828
C03046=1012.207,137.068,-127.585,168.080,77.619,166.735
C03047=1012.207,137.485,-127.621,168.003,77.482,166.636
C03048=1012.208,137.868,-127.654,167.936,77.356,166.548
C03049=1012.208,138.289,-127.690,167.863,77.218,166.452
C03050=1012.208,138.541,-127.712,167.820,77.135,166.395
C03051=1012.208,138.815,-127.736,167.777,77.045,166.336
C03052=1012.208,139.109,-127.762,167.730,76.948,166.272
C03053=1012.208,139.417,-127.788,167.680,76.846,166.205
C03054=1012.209,139.730,-127.815,167.631,76.742,166.139
C03055=1012.208,140.038,-127.842,167.584,76.641,166.074
C03056=1012.209,140.334,-127.867,167.541,76.543,166.014
C03057=1012.209,140.608,-127.891,167.500,76.452,165.958
C03058=1012.208,140.981,-127.923,167.447,76.328,165.884
C03059=1012.209,141.154,-127.939,167.423,76.270,165.849
C03060=1012.209,141.410,-127.961,167.387,76.186,165.799
C03061=1012.210,141.620,-127.979,167.358,76.115,165.758
C03062=1012.209,141.865,-128.000,167.327,76.034,165.712
C03063=1012.210,142.104,-128.020,167.294,75.954,165.665
C03064=1012.210,142.344,-128.041,167.264,75.875,165.621
C03065=1012.210,142.583,-128.062,167.233,75.795,165.576
C03066=1012.210,142.822,-128.083,167.203,75.714,165.532
C03067=1012.210,143.062,-128.104,167.173,75.634,165.488
C03068=1012.210,143.302,-128.125,167.145,75.554,165.445
C03069=1012.211,143.543,-128.145,167.116,75.474,165.402
C03070=1012.211,143.783,-128.167,167.088,75.392,165.359
C03071=1012.212,144.024,-128.187,167.061,75.312,165.318
C03072=1012.211,144.265,-128.208,167.035,75.231,165.276
C03073=1012.211,144.505,-128.229,167.007,75.150,165.234
C03074=1012.212,144.746,-128.250,166.982,75.069,165.193
C03075=1012.212,144.989,-128.271,166.955,74.987,165.152
C03076=1012.213,145.230,-128.292,166.929,74.906,165.111
C03077=1012.213,145.471,-128.312,166.903,74.824,165.071
C03078=1012.213,145.713,-128.334,166.878,74.742,165.031
C03079=1012.213,145.956,-128.355,166.854,74.660,164.991
C03080=1012.214,146.198,-128.376,166.830,74.579,164.953
C03081=1012.214,146.440,-128.397,166.808,74.496,164.915
C03082=1012.214,146.682,-128.418,166.786,74.415,164.877
C03083=1012.215,146.924,-128.440,166.762,74.332,164.838
C03084=1012.215,147.168,-128.460,166.740,74.249,164.800
C03085=1012.215,147.416,-128.482,166.718,74.165,164.762
C03086=1012.215,147.670,-128.504,166.698,74.078,164.724
C03087=1012.216,147.932,-128.527,166.674,73.989,164.684
C03088=1012.216,148.202,-128.550,166.651,73.897,164.644
C03089=1012.217,148.480,-128.575,166.629,73.801,164.603
C03090=1012.217,148.765,-128.599,166.604,73.704,164.560
C03091=1012.218,149.057,-128.625,166.580,73.604,164.517
C03092=1012.218,149.353,-128.651,166.558,73.502,164.475
C03093=1012.219,149.652,-128.677,166.534,73.399,164.432
C03094=1012.219,149.953,-128.703,166.513,73.296,164.390
C03095=1012.220,150.252,-128.729,166.489,73.193,164.347
C03096=1012.220,150.511,-128.752,166.472,73.104,164.312
C03097=1012.221,150.841,-128.781,166.448,72.990,164.266
C03098=1012.221,151.128,-128.806,166.430,72.891,164.228
C03099=1012.222,151.407,-128.829,166.412,72.795,164.191
C03100=1012.223,151.678,-128.853,166.393,72.701,164.154
C03101=1012.222,151.941,-128.876,166.377,72.610,164.120
C03102=1012.223,152.195,-128.898,166.362,72.522,164.087
C03103=1012.224,152.444,-128.921,166.349,72.435,164.055
C03104=1012.224,152.688,-128.941,166.335,72.350,164.024
C03105=1012.225,152.930,-128.963,166.320,72.266,163.993
C03106=1012.226,153.172,-128.984,166.306,72.182,163.962
C03107=1012.226,153.414,-129.005,166.292,72.097,163.931
C03108=1012.227,153.655,-129.026,166.279,72.013,163.900
C03109=1012.226,153.896,-129.047,166.267,71.928,163.871
C03110=1012.227,154.138,-129.068,166.253,71.844,163.840
C03111=1012.228,154.379,-129.089,166.242,71.759,163.812
C03112=1012.229,154.619,-129.110,166.229,71.675,163.782
C03113=1012.229,154.859,-129.131,166.218,71.590,163.753
C03114=1012.230,155.100,-129.152,166.209,71.505,163.725
C03115=1012.231,155.340,-129.174,166.197,71.421,163.696
C03116=1012.230,155.580,-129.194,166.185,71.335,163.667
C03117=1012.231,155.820,-129.215,166.175,71.251,163.639
C03118=1012.232,156.059,-129.236,166.165,71.166,163.611
C03119=1012.233,156.299,-129.257,166.154,71.082,163.583
C03120=1012.233,156.538,-129.278,166.146,70.997,163.556
C03121=1012.234,156.778,-129.299,166.135,70.912,163.528
C03122=1012.235,157.016,-129.320,166.126,70.827,163.501
C03123=1012.236,157.256,-129.341,166.118,70.742,163.474
C03124=1012.236,157.495,-129.362,166.109,70.656,163.447
C03125=1012.237,157.734,-129.383,166.100,70.571,163.420
C03126=1012.237,157.971,-129.404,166.092,70.486,163.394
C03127=1012.238,158.209,-129.424,166.085,70.401,163.368
C03128=1012.239,158.445,-129.445,166.077,70.317,163.342
C03129=1012.240,158.681,-129.466,166.068,70.232,163.315
C03130=1012.240,158.916,-129.486,166.061,70.148,163.290
C03131=1012.241,159.152,-129.507,166.056,70.063,163.265
C03132=1012.242,159.388,-129.527,166.048,69.978,163.240
C03133=1012.242,159.624,-129.549,166.042,69.893,163.215
C03134=1012.244,159.858,-129.569,166.035,69.808,163.190
C03135=1012.244,160.090,-129.589,166.029,69.723,163.165
C03136=1012.244,160.322,-129.612,166.027,69.687,163.155
C03137=1012.243,160.557,-129.637,166.028,69.678,163.153
C03138=1012.243,160.798,-129.661,166.029,69.670,163.151
C03139=1012.243,161.047,-129.687,166.030,69.660,163.149
C03140=1012.242,161.309,-129.714,166.030,69.650,163.147
C03141=1012.241,161.587,-129.743,166.032,69.639,163.145
C03142=1012.240,161.880,-129.773,166.033,69.628,163.142
C03143=1012.240,162.183,-129.804,166.034,69.617,163.140
C03144=1012.239,162.490,-129.836,166.035,69.605,163.137
C03145=1012.239,162.780,-129.866,166.037,69.595,163.135
C03146=1012.238,163.089,-129.898,166.037,69.583,163.133
C03147=1012.237,163.383,-129.929,166.038,69.572,163.130
C03148=1012.237,163.646,-129.955,166.039,69.562,163.128
C03149=1012.236,163.883,-129.980,166.041,69.553,163.127
C03150=1012.236,164.104,-130.003,166.042,69.544,163.125
C03151=1012.234,164.439,-130.038,166.044,69.532,163.123
C03152=1012.234,164.714,-130.066,166.046,69.522,163.121
C03153=1012.234,165.032,-130.099,166.045,69.510,163.118
C03154=1012.233,165.334,-130.130,166.046,69.499,163.115
C03155=1012.233,165.570,-130.155,166.048,69.489,163.114
C03156=1012.232,165.806,-130.179,166.049,69.481,163.112
C03157=1012.231,166.041,-130.204,166.050,69.472,163.111
C03158=1012.231,166.277,-130.228,166.051,69.463,163.109
C03159=1012.230,166.512,-130.253,166.052,69.455,163.107
C03160=1012.230,166.747,-130.278,166.054,69.446,163.106
C03161=1012.230,166.983,-130.302,166.054,69.436,163.103
C03162=1012.229,167.219,-130.327,166.055,69.428,163.101
C03163=1012.229,167.455,-130.351,166.057,69.419,163.100
C03164=1012.228,167.690,-130.376,166.056,69.409,163.097
C03165=1012.227,167.926,-130.400,166.059,69.400,163.096
C03166=1012.227,168.161,-130.425,166.061,69.391,163.095
C03167=1012.226,168.397,-130.449,166.062,69.382,163.093
C03168=1012.226,168.633,-130.474,166.061,69.373,163.090
C03169=1012.225,168.868,-130.498,166.062,69.364,163.089
C03170=1012.226,169.104,-130.523,166.064,69.355,163.087
C03171=1012.224,169.340,-130.547,166.065,69.346,163.086
C03172=1012.224,169.575,-130.572,166.067,69.337,163.084
C03173=1012.224,169.811,-130.596,166.067,69.328,163.082
C03174=1012.223,170.046,-130.621,166.069,69.319,163.080
C03175=1012.223,170.282,-130.646,166.069,69.309,163.078
C03176=1012.222,170.518,-130.669,166.071,69.300,163.077
C03177=1012.222,170.754,-130.695,166.072,69.292,163.075
C03178=1012.221,170.989,-130.719,166.074,69.282,163.074
C03179=1012.221,171.225,-130.744,166.075,69.274,163.072
C03180=1012.220,171.461,-130.768,166.076,69.264,163.070
C03181=1012.220,171.696,-130.793,166.077,69.255,163.068
C03182=1012.219,171.932,-130.818,166.079,69.246,163.067
C03183=1012.219,172.168,-130.842,166.079,69.237,163.064
C03184=1012.220,172.404,-130.867,166.081,69.228,163.063
C03185=1012.218,172.640,-130.891,166.082,69.218,163.061
C03186=1012.218,172.875,-130.916,166.084,69.208,163.059
C03187=1012.217,173.110,-130.941,166.085,69.200,163.058
C03188=1012.217,173.347,-130.965,166.085,69.191,163.055
C03189=1012.217,173.582,-130.990,166.087,69.181,163.054
C03190=1012.216,173.818,-131.015,166.088,69.173,163.052
C03191=1012.216,174.054,-131.039,166.090,69.164,163.051
C03192=1012.215,174.289,-131.065,166.091,69.154,163.049
C03193=1012.215,174.525,-131.089,166.092,69.145,163.047
C03194=1012.214,174.761,-131.114,166.093,69.135,163.045
C03195=1012.214,174.997,-131.138,166.096,69.126,163.044
C03196=1012.215,175.233,-131.163,166.097,69.116,163.042
C03197=1012.213,175.468,-131.188,166.099,69.107,163.040
C03198=1012.213,175.704,-131.212,166.100,69.098,163.039
C03199=1012.212,175.939,-131.237,166.102,69.089,163.037
C03200=1012.213,176.175,-131.262,166.102,69.080,163.035
C03201=1012.212,176.412,-131.287,166.104,69.071,163.034
C03202=1012.211,176.647,-131.311,166.105,69.061,163.032
C03203=1012.211,176.883,-131.335,166.107,69.052,163.030
C03204=1012.211,177.119,-131.361,166.108,69.042,163.028
C03205=1012.211,177.354,-131.386,166.110,69.033,163.027
C03206=1012.210,177.590,-131.410,166.110,69.023,163.024
C03207=1012.210,177.826,-131.435,166.113,69.014,163.023
C03208=1012.210,178.062,-131.460,166.115,69.005,163.022
C03209=1012.209,178.298,-131.484,166.115,68.996,163.019
C03210=1012.208,178.534,-131.510,166.117,68.986,163.018
C03211=1012.209,178.769,-131.534,166.119,68.977,163.017
C03212=1012.207,179.005,-131.559,166.120,68.967,163.015
C03213=1012.208,179.241,-131.584,166.121,68.957,163.013
C03214=1012.207,179.477,-131.609,166.123,68.948,163.012
C03215=1012.207,179.713,-131.633,166.124,68.938,163.009
C03216=1012.206,179.948,-131.658,166.127,68.929,163.008
C03217=1012.206,180.184,-131.683,166.128,68.919,163.006
C03218=1012.206,180.420,-131.709,166.129,68.911,163.005
C03219=1012.206,180.656,-131.733,166.131,68.902,163.003
C03220=1012.205,180.892,-131.758,166.132,68.892,163.001
C03221=1012.205,181.127,-131.783,166.134,68.883,163.000
C03222=1012.204,181.364,-131.808,166.135,68.873,162.998
C03223=1012.204,181.599,-131.832,166.138,68.864,162.997
C03224=1012.204,181.835,-131.858,166.139,68.854,162.995
C03225=1012.204,182.072,-131.882,166.140,68.844,162.993
C03226=1012.203,182.307,-131.907,166.142,68.835,162.991
C03227=1012.203,182.542,-131.932,166.143,68.825,162.989
C03228=1012.203,182.778,-131.957,166.145,68.816,162.988
C03229=1012.203,183.015,-131.982,166.148,68.807,162.987
C03230=1012.202,183.251,-132.007,166.149,68.797,162.985
C03231=1012.202,183.486,-132.032,166.151,68.788,162.984
C03232=1012.202,183.722,-132.057,166.152,68.778,162.982
C03233=1012.201,183.958,-132.081,166.153,68.768,162.980
C03234=1012.201,184.194,-132.107,166.156,68.759,162.978
C03235=1012.201,184.429,-132.131,166.158,68.748,162.977
C03236=1012.201,184.665,-132.157,166.159,68.738,162.975
C03237=1012.200,184.902,-132.182,166.161,68.729,162.973
C03238=1012.200,185.138,-132.207,166.163,68.720,162.972
C03239=1012.200,185.374,-132.232,166.165,68.710,162.970
C03240=1012.200,185.609,-132.257,166.167,68.701,162.969
C03241=1012.199,185.845,-132.282,166.168,68.691,162.967
C03242=1012.199,186.082,-132.306,166.169,68.681,162.965
C03243=1012.198,186.317,-132.332,166.171,68.672,162.964
C03244=1012.199,186.552,-132.356,166.174,68.662,162.962
C03245=1012.198,186.788,-132.382,166.175,68.652,162.960
C03246=1012.198,187.024,-132.407,166.177,68.643,162.959
C03247=1012.198,187.261,-132.431,166.178,68.633,162.957
C03248=1012.197,187.497,-132.457,166.181,68.624,162.956
C03249=1012.197,187.732,-132.482,166.182,68.614,162.954
C03250=1012.197,187.968,-132.507,166.184,68.605,162.952
C03251=1012.197,188.204,-132.532,166.186,68.594,162.951
C03252=1012.196,188.440,-132.557,166.188,68.584,162.949
C03253=1012.196,188.676,-132.582,166.190,68.575,162.948
C03254=1012.196,188.912,-132.607,166.192,68.565,162.946
C03255=1012.196,189.148,-132.633,166.193,68.555,162.944
C03256=1012.196,189.384,-132.657,166.195,68.545,162.942
C03257=1012.195,189.620,-132.683,166.198,68.535,162.941
C03258=1012.195,189.856,-132.708,166.200,68.526,162.940
C03259=1012.195,190.092,-132.733,166.202,68.517,162.938
C03260=1012.194,190.328,-132.758,166.203,68.507,162.936
C03261=1012.195,190.564,-132.783,166.206,68.497,162.935
C03262=1012.194,190.800,-132.808,166.208,68.487,162.933
C03263=1012.194,191.035,-132.834,166.210,68.477,162.932
C03264=1012.195,191.272,-132.859,166.211,68.467,162.930
C03265=1012.194,191.508,-132.884,166.213,68.456,162.928
C03266=1012.194,191.743,-132.909,166.216,68.447,162.927
C03267=1012.194,191.979,-132.935,166.218,68.438,162.926
C03268=1012.193,192.215,-132.960,166.219,68.428,162.924
C03269=1012.193,192.452,-132.984,166.222,68.418,162.922
C03270=1012.193,192.688,-133.010,166.224,68.409,162.921
C03271=1012.193,192.923,-133.035,166.225,68.399,162.919
C03272=1012.193,193.159,-133.060,166.228,68.389,162.918
C03273=1012.192,193.395,-133.086,166.230,68.378,162.916
C03274=1012.193,193.632,-133.111,166.231,68.368,162.914
C03275=1012.193,193.868,-133.136,166.235,68.359,162.913
C03276=1012.192,194.104,-133.162,166.236,68.349,162.912
C03277=1012.192,194.339,-133.187,166.239,68.340,162.910
C03278=1012.192,194.575,-133.212,166.241,68.329,162.909
C03279=1012.192,194.811,-133.237,166.242,68.319,162.907
C03280=1012.192,195.047,-133.262,166.246,68.310,162.906
C03281=1012.192,195.283,-133.288,166.247,68.300,162.904
C03282=1012.192,195.519,-133.313,166.249,68.290,162.903
C03283=1012.192,195.755,-133.339,166.252,68.279,162.901
C03284=1012.191,195.991,-133.364,166.254,68.269,162.899
C03285=1012.191,196.227,-133.389,166.255,68.259,162.898
C03286=1012.191,196.463,-133.414,166.259,68.249,162.897
C03287=1012.191,196.699,-133.440,166.260,68.239,162.895
C03288=1012.191,196.935,-133.465,166.263,68.230,162.894
C03289=1012.191,197.171,-133.490,166.265,68.220,162.892
C03290=1012.191,197.407,-133.515,166.268,68.210,162.891
C03291=1012.191,197.643,-133.541,166.270,68.201,162.889
C03292=1012.191,197.879,-133.567,166.272,68.190,162.888
C03293=1012.191,198.115,-133.592,166.275,68.180,162.886
C03294=1012.191,198.351,-133.617,166.277,68.169,162.885
C03295=1012.191,198.598,-133.644,166.280,68.159,162.883
C03296=1012.190,198.989,-133.686,166.282,68.142,162.880
C03297=1012.191,199.380,-133.729,166.286,68.126,162.878
C03298=1012.190,199.622,-133.754,166.290,68.115,162.877
C03299=1012.190,199.851,-133.778,166.292,68.106,162.875
C03300=1012.191,200.084,-133.803,166.295,68.095,162.874
C03301=1012.191,200.326,-133.830,166.297,68.085,162.872
C03302=1012.190,200.579,-133.858,166.299,68.075,162.871
C03303=1012.190,200.835,-133.885,166.302,68.063,162.869
C03304=1012.191,201.074,-133.911,166.304,68.052,162.867
C03305=1012.191,201.296,-133.935,166.307,68.043,162.866
C03306=1012.190,201.513,-133.959,166.309,68.034,162.865
C03307=1012.191,201.930,-134.004,166.314,68.016,162.863
C03308=1012.191,202.136,-134.025,166.316,68.008,162.861
C03309=1012.191,202.354,-134.049,166.317,67.998,162.859
C03310=1012.196,203.604,-134.186,167.164,68.086,163.263
C03311=1012.198,203.850,-134.213,167.166,68.075,163.261
C03312=1012.200,204.093,-134.239,167.170,68.066,163.260
C03313=1012.202,204.336,-134.266,167.173,68.056,163.259
C03314=1012.205,204.581,-134.292,167.175,68.046,163.257
C03315=1012.207,204.825,-134.319,167.178,68.036,163.256
C03316=1012.209,205.069,-134.345,167.181,68.026,163.254
C03317=1012.212,205.313,-134.372,167.183,68.017,163.253
C03318=1012.214,205.558,-134.398,167.186,68.007,163.252
C03319=1012.215,205.801,-134.425,167.188,67.997,163.250
C03320=1012.218,206.045,-134.452,167.191,67.987,163.249
C03321=1012.220,206.289,-134.478,167.195,67.977,163.248
C03322=1012.222,206.533,-134.505,167.197,67.967,163.246
C03323=1012.225,206.776,-134.531,167.200,67.958,163.245
C03324=1012.227,207.018,-134.558,167.204,67.948,163.244
C03325=1012.229,207.261,-134.584,167.206,67.938,163.242
C03326=1012.232,207.504,-134.611,167.209,67.928,163.241
C03327=1012.234,207.747,-134.637,167.212,67.918,163.240
C03328=1012.237,207.990,-134.664,167.216,67.909,163.239
C03329=1012.238,208.232,-134.690,167.218,67.898,163.237
C03330=1012.240,208.475,-134.716,167.220,67.889,163.235
C03331=1012.243,208.718,-134.744,167.223,67.880,163.234
C03332=1012.245,208.961,-134.770,167.227,67.870,163.233
C03333=1012.247,209.202,-134.796,167.230,67.861,163.232
C03334=1012.250,209.445,-134.822,167.232,67.850,163.230
C03335=1012.252,209.688,-134.849,167.236,67.841,163.229
C03336=1012.254,209.930,-134.876,167.238,67.832,163.228
C03337=1012.257,210.172,-134.902,167.241,67.822,163.227
C03338=1012.259,210.415,-134.929,167.243,67.812,163.225
C03339=1012.261,210.657,-134.955,167.247,67.802,163.224
C03340=1012.264,210.900,-134.982,167.250,67.792,163.223
C03341=1012.266,211.143,-135.009,167.253,67.783,163.222
C03342=1012.268,211.385,-135.036,167.257,67.773,163.220
C03343=1012.271,211.628,-135.062,167.258,67.764,163.218
C03344=1012.273,211.871,-135.088,167.261,67.754,163.217
C03345=1012.275,212.114,-135.115,167.265,67.744,163.216
C03346=1012.278,212.358,-135.142,167.268,67.735,163.215
C03347=1012.280,212.601,-135.169,167.271,67.725,163.214
C03348=1012.282,212.844,-135.195,167.275,67.716,163.213
C03349=1012.285,213.088,-135.222,167.278,67.706,163.212
C03350=1012.287,213.332,-135.249,167.279,67.696,163.210
C03351=1012.290,213.575,-135.276,167.283,67.687,163.209
C03352=1012.292,213.820,-135.303,167.286,67.677,163.208
C03353=1012.295,214.064,-135.330,167.289,67.667,163.206
C03354=1012.297,214.308,-135.356,167.293,67.658,163.205
C03355=1012.300,214.553,-135.384,167.296,67.648,163.204
C03356=1012.302,214.797,-135.410,167.299,67.639,163.203
C03357=1012.304,215.042,-135.438,167.302,67.630,163.202
C03358=1012.307,215.287,-135.464,167.305,67.620,163.201
C03359=1012.310,215.533,-135.491,167.307,67.610,163.199
C03360=1012.312,215.778,-135.518,167.311,67.600,163.198
C03361=1012.314,216.024,-135.545,167.314,67.591,163.197
C03362=1012.317,216.269,-135.572,167.318,67.581,163.196
C03363=1012.320,216.515,-135.599,167.321,67.572,163.195
C03364=1012.322,216.761,-135.626,167.324,67.562,163.194
C03365=1012.324,217.009,-135.654,167.328,67.552,163.192
C03366=1012.328,217.264,-135.682,167.330,67.542,163.191
C03367=1012.330,217.524,-135.711,167.333,67.533,163.190
C03368=1012.333,217.788,-135.740,167.337,67.522,163.188
C03369=1012.335,218.069,-135.771,167.340,67.511,163.187
C03370=1012.338,218.358,-135.804,167.344,67.500,163.185
C03371=1012.342,218.651,-135.836,167.348,67.488,163.184
C03372=1012.345,218.948,-135.869,167.353,67.477,163.183
C03373=1012.348,219.252,-135.903,167.357,67.466,163.182
C03374=1012.351,219.548,-135.935,167.361,67.455,163.181
C03375=1012.354,219.829,-135.966,167.365,67.443,163.180
C03376=1012.357,220.101,-135.997,167.369,67.434,163.179
C03377=1012.359,220.362,-136.026,167.372,67.423,163.177
C03378=1012.362,220.611,-136.054,167.374,67.414,163.176
C03379=1012.365,220.857,-136.081,167.378,67.404,163.175
C03380=1012.367,221.103,-136.108,167.381,67.395,163.174
C03381=1012.371,221.349,-136.135,167.385,67.385,163.173
C03382=1012.373,221.594,-136.163,167.388,67.376,163.171
C03383=1012.376,221.840,-136.190,167.390,67.367,163.170
C03384=1012.378,222.085,-136.217,167.395,67.358,163.170
C03385=1012.381,222.332,-136.245,167.397,67.349,163.168
C03386=1012.384,222.578,-136.272,167.401,67.339,163.167
C03387=1012.386,222.823,-136.300,167.405,67.331,163.167
C03388=1012.389,223.069,-136.327,167.407,67.322,163.165
C03389=1012.391,223.314,-136.355,167.411,67.312,163.164
C03390=1012.394,223.561,-136.382,167.414,67.303,163.163
C03391=1012.397,223.807,-136.409,167.418,67.293,163.162
C03392=1012.399,224.052,-136.437,167.421,67.283,163.161
C03393=1012.403,224.298,-136.464,167.425,67.274,163.160
C03394=1012.406,224.544,-136.492,167.428,67.264,163.159
C03395=1012.408,224.789,-136.519,167.430,67.255,163.158
C03396=1012.411,225.035,-136.547,167.435,67.247,163.157
C03397=1012.413,225.281,-136.574,167.437,67.238,163.156
C03398=1012.416,225.527,-136.601,167.441,67.228,163.155
C03399=1012.419,225.772,-136.630,167.445,67.219,163.154
C03400=1012.422,226.018,-136.657,167.449,67.210,163.153
C03401=1012.424,226.264,-136.684,167.451,67.201,163.152
C03402=1012.427,226.510,-136.712,167.455,67.191,163.151
C03403=1012.430,226.755,-136.739,167.458,67.182,163.150
C03404=1012.433,227.000,-136.767,167.463,67.172,163.149
C03405=1012.436,227.247,-136.794,167.465,67.163,163.148
C03406=1012.438,227.492,-136.821,167.470,67.154,163.147
C03407=1012.442,227.738,-136.850,167.472,67.145,163.146
C03408=1012.444,227.984,-136.877,167.476,67.136,163.146
C03409=1012.448,228.230,-136.905,167.479,67.127,163.144
C03410=1012.450,228.475,-136.932,167.483,67.118,163.144
C03411=1012.453,228.721,-136.960,167.487,67.109,163.143
C03412=1012.456,228.967,-136.988,167.490,67.099,163.142
C03413=1012.458,229.212,-137.016,167.493,67.090,163.140
C03414=1012.462,229.458,-137.043,167.496,67.081,163.139
C03415=1012.465,229.703,-137.071,167.500,67.071,163.138
C03416=1012.468,229.950,-137.098,167.504,67.063,163.138
C03417=1012.470,230.195,-137.126,167.507,67.054,163.136
C03418=1012.473,230.441,-137.153,167.511,67.045,163.136
C03419=1012.476,230.686,-137.182,167.514,67.036,163.135
C03420=1012.479,230.933,-137.209,167.518,67.027,163.134
C03421=1012.481,231.177,-137.237,167.520,67.018,163.133
C03422=1012.485,231.423,-137.265,167.525,67.009,163.132
C03423=1012.487,231.669,-137.292,167.529,67.000,163.131
C03424=1012.491,231.915,-137.320,167.532,66.990,163.130
C03425=1012.494,232.161,-137.348,167.536,66.981,163.129
C03426=1012.496,232.406,-137.375,167.539,66.971,163.128
C03427=1012.500,232.651,-137.403,167.543,66.963,163.127
C03428=1012.502,232.897,-137.431,167.546,66.955,163.127
C03429=1012.506,233.143,-137.459,167.551,66.946,163.126
C03430=1012.509,233.389,-137.487,167.553,66.937,163.125
C03431=1012.511,233.634,-137.515,167.558,66.929,163.125
C03432=1012.514,233.880,-137.543,167.561,66.919,163.124
C03433=1012.517,234.125,-137.571,167.563,66.910,163.122
C03434=1012.521,234.371,-137.598,167.568,66.901,163.122
C03435=1012.524,234.617,-137.626,167.572,66.892,163.121
C03436=1012.527,234.863,-137.654,167.575,66.882,163.120
C03437=1012.529,235.107,-137.682,167.579,66.873,163.119
C03438=1012.532,235.353,-137.710,167.582,66.865,163.118
C03439=1012.536,235.599,-137.738,167.586,66.857,163.117
C03440=1012.538,235.845,-137.765,167.590,66.848,163.117
C03441=1012.542,236.090,-137.794,167.594,66.840,163.116
C03442=1012.545,236.336,-137.822,167.597,66.830,163.115
C03443=1012.548,236.581,-137.849,167.601,66.822,163.114
C03444=1012.551,236.826,-137.877,167.604,66.812,163.113
C03445=1012.554,237.072,-137.905,167.609,66.804,163.113
C03446=1012.557,237.317,-137.934,167.612,66.794,163.112
C03447=1012.560,237.563,-137.962,167.616,66.785,163.111
C03448=1012.563,237.809,-137.989,167.619,66.776,163.110
C03449=1012.566,238.055,-138.017,167.623,66.768,163.109
C03450=1012.569,238.300,-138.046,167.627,66.760,163.109
C03451=1012.572,238.546,-138.074,167.631,66.751,163.108
C03452=1012.576,238.792,-138.102,167.633,66.742,163.107
C03453=1012.579,239.037,-138.129,167.638,66.734,163.106
C03454=1012.583,239.282,-138.158,167.642,66.725,163.106
C03455=1012.586,239.528,-138.186,167.645,66.716,163.105
C03456=1012.588,239.773,-138.214,167.648,66.707,163.104
C03457=1012.591,240.019,-138.242,167.653,66.698,163.103
C03458=1012.594,240.264,-138.270,167.657,66.688,163.102
C03459=1012.598,240.510,-138.298,167.660,66.680,163.101
C03460=1012.601,240.755,-138.326,167.664,66.672,163.101
C03461=1012.604,241.000,-138.355,167.668,66.663,163.100
C03462=1012.607,241.246,-138.383,167.672,66.655,163.100
C03463=1012.611,241.491,-138.411,167.675,66.647,163.099
C03464=1012.614,241.737,-138.439,167.680,66.638,163.099
C03465=1012.617,241.982,-138.467,167.683,66.629,163.097
C03466=1012.620,242.228,-138.495,167.687,66.621,163.097
C03467=1012.623,242.474,-138.524,167.690,66.611,163.096
C03468=1012.627,242.719,-138.552,167.695,66.602,163.095
C03469=1012.630,242.964,-138.581,167.699,66.593,163.094
C03470=1012.633,243.210,-138.609,167.702,66.585,163.094
C03471=1012.636,243.455,-138.637,167.707,66.577,163.093
C03472=1012.639,243.701,-138.665,167.710,66.569,163.093
C03473=1012.644,243.946,-138.693,167.714,66.561,163.092
C03474=1012.647,244.192,-138.722,167.718,66.552,163.092
C03475=1012.650,244.438,-138.750,167.721,66.543,163.090
C03476=1012.653,244.683,-138.778,167.725,66.535,163.090
C03477=1012.657,244.928,-138.807,167.730,66.526,163.089
C03478=1012.660,245.174,-138.835,167.734,66.516,163.088
C03479=1012.663,245.419,-138.863,167.737,66.508,163.088
C03480=1012.666,245.665,-138.892,167.742,66.500,163.087
C03481=1012.670,245.910,-138.921,167.745,66.491,163.087
C03482=1012.673,246.155,-138.949,167.749,66.483,163.086
C03483=1012.676,246.400,-138.978,167.752,66.475,163.085
C03484=1012.680,246.646,-139.005,167.757,66.466,163.085
C03485=1012.683,246.891,-139.033,167.760,66.458,163.084
C03486=1012.687,247.137,-139.063,167.764,66.450,163.083
C03487=1012.690,247.383,-139.091,167.769,66.441,163.083
///RCONF 0,0,0,0,1,0,0,0,0,0,0,0,0,0,0,0,0,0,0,0,0,0,0,0
C03488=1012.694,247.628,-139.120,167.773,66.433,163.082
C03489=1012.697,247.873,-139.148,167.777,66.423,163.081
C03490=1012.700,248.119,-139.176,167.781,66.414,163.081
C03491=1012.703,248.364,-139.205,167.784,66.407,163.080
C03492=1012.706,248.609,-139.233,167.789,66.398,163.080
C03493=1012.710,248.855,-139.262,167.793,66.391,163.079
C03494=1012.714,249.101,-139.290,167.797,66.383,163.079
C03495=1012.717,249.346,-139.319,167.800,66.374,163.078
C03496=1012.721,249.591,-139.347,167.805,66.366,163.078
C03497=1012.724,249.836,-139.376,167.808,66.358,163.077
C03498=1012.728,250.082,-139.405,167.813,66.349,163.076
C03499=1012.731,250.327,-139.433,167.815,66.340,163.075
C03500=1012.735,250.572,-139.462,167.820,66.331,163.075
C03501=1012.738,250.818,-139.490,167.825,66.323,163.074
C03502=1012.741,251.063,-139.519,167.828,66.314,163.074
C03503=1012.745,251.308,-139.548,167.833,66.307,163.073
C03504=1012.749,251.554,-139.577,167.836,66.299,163.073
C03505=1012.752,251.799,-139.605,167.841,66.291,163.073
C03506=1012.755,252.044,-139.634,167.845,66.283,163.072
C03507=1012.759,252.290,-139.663,167.849,66.275,163.072
C03508=1012.763,252.535,-139.692,167.853,66.267,163.071
C03509=1012.766,252.780,-139.721,167.857,66.258,163.070
C03510=1012.770,253.025,-139.748,167.861,66.248,163.069
C03511=1012.774,253.271,-139.777,167.865,66.240,163.069
C03512=1012.777,253.516,-139.806,167.869,66.232,163.068
C03513=1012.781,253.761,-139.835,167.874,66.224,163.068
C03514=1012.784,254.007,-139.864,167.877,66.216,163.067
C03515=1012.788,254.252,-139.893,167.882,66.209,163.067
C03516=1012.791,254.497,-139.921,167.885,66.200,163.067
C03517=1012.795,254.742,-139.950,167.890,66.193,163.066
C03518=1012.799,254.988,-139.980,167.895,66.184,163.066
C03519=1012.802,255.234,-140.008,167.898,66.176,163.065
C03520=1012.805,255.479,-140.037,167.903,66.168,163.065
C03521=1012.809,255.724,-140.066,167.905,66.159,163.064
C03522=1012.813,255.969,-140.095,167.910,66.150,163.063
C03523=1012.817,256.215,-140.124,167.915,66.143,163.063
C03524=1012.820,256.460,-140.153,167.918,66.135,163.062
C03525=1012.823,256.705,-140.182,167.923,66.127,163.062
C03526=1012.828,256.951,-140.211,167.927,66.120,163.062
C03527=1012.831,257.196,-140.240,167.931,66.112,163.061
C03528=1012.834,257.440,-140.269,167.936,66.103,163.061
C03529=1012.838,257.686,-140.298,167.940,66.096,163.061
C03530=1012.843,257.931,-140.326,167.945,66.087,163.060
C03531=1012.847,258.177,-140.356,167.948,66.079,163.060
C03532=1012.850,258.421,-140.385,167.952,66.069,163.059
C03533=1012.853,258.666,-140.413,167.957,66.061,163.058
C03534=1012.868,259.922,-140.569,167.736,65.990,162.948
C03535=1012.870,260.336,-140.624,167.663,65.983,162.916
C03536=1012.872,260.751,-140.679,167.588,65.941,162.874
C03537=1012.874,261.165,-140.736,167.513,65.920,162.838
C03538=1012.873,261.579,-140.795,167.439,65.902,162.803
C03539=1012.873,261.994,-140.853,167.365,65.851,162.759
C03540=1012.870,262.408,-140.915,167.291,65.835,162.724
C03541=1012.868,262.822,-140.977,167.217,65.802,162.686
C03542=1012.863,263.237,-141.042,167.142,65.796,162.653
C03543=1012.858,263.651,-141.107,167.067,65.756,162.613
C03544=1012.853,264.065,-141.175,166.991,65.747,162.580
C03545=1012.845,264.479,-141.243,166.916,65.725,162.544
///RCONF 0,0,0,0,0,0,0,0,0,0,0,0,0,0,0,0,0,0,0,0,0,0,0,0
C03546=1012.838,264.892,-141.313,166.845,65.678,162.503
C03547=1012.828,265.306,-141.385,166.768,65.679,162.472
C03548=1012.818,265.720,-141.457,166.693,65.647,162.433
C03549=1012.808,266.133,-141.531,166.619,65.612,162.395
C03550=1012.796,266.546,-141.606,166.544,65.589,162.359
C03551=1012.782,266.959,-141.685,166.467,65.575,162.325
C03552=1012.768,267.372,-141.762,166.393,65.555,162.290
C03553=1012.753,267.785,-141.842,166.320,65.521,162.252
C03554=1012.737,268.197,-141.925,166.240,65.519,162.219
C03555=1012.720,268.610,-142.007,166.167,65.483,162.182
C03556=1012.702,269.023,-142.092,166.091,65.464,162.147
C03557=1012.683,269.435,-142.178,166.013,65.452,162.113
C03558=1012.663,269.847,-142.264,165.943,65.406,162.073
C03559=1012.641,270.258,-142.354,165.865,65.392,162.039
C03560=1012.620,270.670,-142.443,165.791,65.361,162.002
C03561=1012.596,271.082,-142.536,165.710,65.360,161.970
C03562=1012.572,271.494,-142.628,165.638,65.324,161.933
